LIN {X 0,Y 346.916,Z 553.438,A -85,B 0,C 180,E1 16644.293,E2 16644.293} C_VEL
LIN {X 0,Y 348.339,Z 562.311,A -85,B 0,C 180,E1 16644.634,E2 16644.634} C_VEL
LIN {X 0,Y 348.733,Z 569.969,A -85,B 0,C 180,E1 16644.843,E2 16644.843} C_VEL
LIN {X 0,Y 347.091,Z 583.273,A -85,B 0,C 180,E1 16645.017,E2 16645.017} C_VEL
LIN {X 0,Y 345.326,Z 596.669,A -85,B 0,C 180,E1 16645.186,E2 16645.186} C_VEL
LIN {X 0,Y 345.275,Z 597.789,A -85,B 0,C 180,E1 16645.208,E2 16645.208} C_VEL
LIN {X 0,Y 342.847,Z 683.726,A -85,B 0,C 180,E1 16647.121,E2 16647.121} C_VEL
LIN {X 0,Y 342.056,Z 700.444,A -85,B 0,C 180,E1 16647.822,E2 16647.822} C_VEL
LIN {X 0,Y 340.975,Z 714.968,A -85,B 0,C 180,E1 16648.731,E2 16648.731} C_VEL
LIN {X 0,Y 339.513,Z 729.938,A -85,B 0,C 180,E1 16650,E2 16650} C_VEL
LIN {X 0,Y 337.856,Z 743.563,A -85,B 0,C 180,E1 16651.526,E2 16651.526} C_VEL
LIN {X 0,Y 336.233,Z 755.603,A -85,B 0,C 180,E1 16653.239,E2 16653.239} C_VEL
LIN {X 0,Y 334.524,Z 767.051,A -85,B 0,C 180,E1 16655.316,E2 16655.316} C_VEL
LIN {X 0,Y 333.111,Z 776.185,A -85,B 0,C 180,E1 16657.415,E2 16657.415} C_VEL
LIN {X 0,Y 331.821,Z 784.518,A -85,B 0,C 180,E1 16659.89,E2 16659.89} C_VEL
LIN {X 0,Y 330.892,Z 790.802,A -85,B 0,C 180,E1 16662.388,E2 16662.388} C_VEL
LIN {X 0,Y 330.281,Z 795.59,A -85,B 0,C 180,E1 16665.09,E2 16665.09} C_VEL
LIN {X 0,Y 330.001,Z 798.505,A -85,B 0,C 180,E1 16667.819,E2 16667.819} C_VEL
LIN {X 0,Y 330.029,Z 799.71,A -85,B 0,C 180,E1 16670.584,E2 16670.584} C_VEL
LIN {X 0,Y 330.354,Z 799.125,A -85,B 0,C 180,E1 16673.359,E2 16673.359} C_VEL
LIN {X 0,Y 331.055,Z 796.754,A -85,B 0,C 180,E1 16676.164,E2 16676.164} C_VEL
LIN {X 0,Y 332.129,Z 792.619,A -85,B 0,C 180,E1 16678.83,E2 16678.83} C_VEL
LIN {X 0,Y 333.632,Z 786.717,A -85,B 0,C 180,E1 16681.43,E2 16681.43} C_VEL
LIN {X 0,Y 335.47,Z 779.072,A -85,B 0,C 180,E1 16683.872,E2 16683.872} C_VEL
LIN {X 0,Y 337.579,Z 769.937,A -85,B 0,C 180,E1 16686.115,E2 16686.115} C_VEL
LIN {X 0,Y 339.943,Z 758.678,A -85,B 0,C 180,E1 16688.249,E2 16688.249} C_VEL
LIN {X 0,Y 342.175,Z 746.843,A -85,B 0,C 180,E1 16690.005,E2 16690.005} C_VEL
LIN {X 0,Y 344.428,Z 733.255,A -85,B 0,C 180,E1 16691.58,E2 16691.58} C_VEL
LIN {X 0,Y 346.309,Z 719.123,A -85,B 0,C 180,E1 16692.832,E2 16692.832} C_VEL
LIN {X 0,Y 347.866,Z 703.791,A -85,B 0,C 180,E1 16693.844,E2 16693.844} C_VEL
LIN {X 0,Y 348.904,Z 687.638,A -85,B 0,C 180,E1 16694.564,E2 16694.564} C_VEL
LIN {X 0,Y 349.945,Z 659.796,A -85,B 0,C 180,E1 16695.275,E2 16695.275} C_VEL
LIN {X 0,Y 352.345,Z 591.836,A -85,B 0,C 180,E1 16696.795,E2 16696.795} C_VEL
LIN {X 0,Y 347.322,Z 564.262,A -85,B 0,C 180,E1 16698.138,E2 16698.138} C_VEL
LIN {X 0,Y 345.002,Z 552.728,A -85,B 0,C 180,E1 16698.806,E2 16698.806} C_VEL
LIN {X 0,Y 349.556,Z 526.788,A -85,B 0,C 180,E1 16703.353,E2 16703.353} C_VEL
LIN {X 0,Y 350.462,Z 522.011,A -85,B 0,C 180,E1 16704.206,E2 16704.206} C_VEL
LIN {X 0,Y 347.626,Z 509.823,A -85,B 0,C 180,E1 16707.266,E2 16707.266} C_VEL
LIN {X 0,Y 344.077,Z 497.71,A -85,B 0,C 180,E1 16710.665,E2 16710.665} C_VEL
LIN {X 0,Y 340.458,Z 487.061,A -85,B 0,C 180,E1 16714.05,E2 16714.05} C_VEL
LIN {X 0,Y 336.824,Z 477.501,A -85,B 0,C 180,E1 16717.484,E2 16717.484} C_VEL
LIN {X 0,Y 333.454,Z 469.646,A -85,B 0,C 180,E1 16720.741,E2 16720.741} C_VEL
LIN {X 0,Y 331.399,Z 465.22,A -85,B 0,C 180,E1 16722.802,E2 16722.802} C_VEL
LIN {X 0,Y 330.06,Z 461.809,A -85,B 0,C 180,E1 16724.539,E2 16724.539} C_VEL
LIN {X 0,Y 330.044,Z 461.676,A -85,B 0,C 180,E1 16728.82,E2 16728.82} C_VEL
LIN {X 0,Y 330.056,Z 461.676,A -85,B 0,C 180,E1 16733.215,E2 16733.215} C_VEL
LIN {X 0,Y 330.051,Z 461.685,A -85,B 0,C 180,E1 16737.569,E2 16737.569} C_VEL
LIN {X 0,Y 330.049,Z 461.686,A -85,B 0,C 180,E1 16741.909,E2 16741.909} C_VEL
LIN {X 0,Y 330.05,Z 461.673,A -85,B 0,C 180,E1 16746.261,E2 16746.261} C_VEL
LIN {X 0,Y 330.04,Z 461.665,A -85,B 0,C 180,E1 16750.649,E2 16750.649} C_VEL
LIN {X 0,Y 330.041,Z 461.658,A -85,B 0,C 180,E1 16754.922,E2 16754.922} C_VEL
LIN {X 0,Y 330.044,Z 461.659,A -85,B 0,C 180,E1 16759.281,E2 16759.281} C_VEL
LIN {X 0,Y 330.048,Z 461.661,A -85,B 0,C 180,E1 16763.571,E2 16763.571} C_VEL
LIN {X 0,Y 330.052,Z 461.662,A -85,B 0,C 180,E1 16768.005,E2 16768.005} C_VEL
LIN {X 0,Y 330.104,Z 462.019,A -85,B 0,C 180,E1 16770.785,E2 16770.785} C_VEL
LIN {X 0,Y 331.718,Z 465.65,A -85,B 0,C 180,E1 16772.447,E2 16772.447} C_VEL
LIN {X 0,Y 332.9,Z 468.27,A -85,B 0,C 180,E1 16773.548,E2 16773.548} C_VEL
LIN {X 0,Y 334.783,Z 471.961,A -85,B 0,C 180,E1 16775.083,E2 16775.083} C_VEL
LIN {X 0,Y 336.969,Z 476.649,A -85,B 0,C 180,E1 16776.825,E2 16776.825} C_VEL
LIN {X 0,Y 340.192,Z 483.549,A -85,B 0,C 180,E1 16779.191,E2 16779.191} C_VEL
LIN {X 0,Y 344.869,Z 494.751,A -85,B 0,C 180,E1 16782.494,E2 16782.494} C_VEL
LIN {X 0,Y 349.82,Z 507.787,A -85,B 0,C 180,E1 16785.781,E2 16785.781} C_VEL
LIN {X 0,Y 354.514,Z 522.198,A -85,B 0,C 180,E1 16788.918,E2 16788.918} C_VEL
LIN {X 0,Y 355.858,Z 526.854,A -85,B 0,C 180,E1 16789.839,E2 16789.839} C_VEL
LIN {X 0,Y 352.603,Z 543.562,A -85,B 0,C 180,E1 16791.896,E2 16791.896} C_VEL
LIN {X 0,Y 355.658,Z 572.916,A -85,B 0,C 180,E1 16793.022,E2 16793.022} C_VEL
LIN {X 0,Y 350.526,Z 732.105,A -85,B 0,C 180,E1 16796.34,E2 16796.34} C_VEL
LIN {X 0,Y 349.044,Z 750.459,A -85,B 0,C 180,E1 16796.989,E2 16796.989} C_VEL
LIN {X 0,Y 346.94,Z 768.318,A -85,B 0,C 180,E1 16797.918,E2 16797.918} C_VEL
LIN {X 0,Y 344.525,Z 784.972,A -85,B 0,C 180,E1 16799.091,E2 16799.091} C_VEL
LIN {X 0,Y 341.851,Z 801.23,A -85,B 0,C 180,E1 16800.569,E2 16800.569} C_VEL
LIN {X 0,Y 339.127,Z 816.442,A -85,B 0,C 180,E1 16802.305,E2 16802.305} C_VEL
LIN {X 0,Y 336.369,Z 831.077,A -85,B 0,C 180,E1 16804.365,E2 16804.365} C_VEL
LIN {X 0,Y 333.867,Z 844.636,A -85,B 0,C 180,E1 16806.715,E2 16806.715} C_VEL
LIN {X 0,Y 331.697,Z 857.019,A -85,B 0,C 180,E1 16809.349,E2 16809.349} C_VEL
LIN {X 0,Y 330.098,Z 867.902,A -85,B 0,C 180,E1 16812.186,E2 16812.186} C_VEL
LIN {X 0,Y 329.089,Z 877.24,A -85,B 0,C 180,E1 16815.214,E2 16815.214} C_VEL
LIN {X 0,Y 328.711,Z 884.849,A -85,B 0,C 180,E1 16818.362,E2 16818.362} C_VEL
LIN {X 0,Y 328.8,Z 890.405,A -85,B 0,C 180,E1 16821.431,E2 16821.431} C_VEL
LIN {X 0,Y 329.17,Z 894.144,A -85,B 0,C 180,E1 16824.422,E2 16824.422} C_VEL
LIN {X 0,Y 329.528,Z 896.232,A -85,B 0,C 180,E1 16827.392,E2 16827.392} C_VEL
LIN {X 0,Y 329.683,Z 896.689,A -85,B 0,C 180,E1 16830.174,E2 16830.174} C_VEL
LIN {X 0,Y 329.551,Z 895.671,A -85,B 0,C 180,E1 16832.957,E2 16832.957} C_VEL
LIN {X 0,Y 329.242,Z 893.161,A -85,B 0,C 180,E1 16835.752,E2 16835.752} C_VEL
LIN {X 0,Y 328.911,Z 888.783,A -85,B 0,C 180,E1 16838.743,E2 16838.743} C_VEL
LIN {X 0,Y 328.841,Z 882.577,A -85,B 0,C 180,E1 16841.755,E2 16841.755} C_VEL
LIN {X 0,Y 329.177,Z 874.384,A -85,B 0,C 180,E1 16844.783,E2 16844.783} C_VEL
LIN {X 0,Y 330.035,Z 864.634,A -85,B 0,C 180,E1 16847.636,E2 16847.636} C_VEL
LIN {X 0,Y 331.368,Z 853.376,A -85,B 0,C 180,E1 16850.304,E2 16850.304} C_VEL
LIN {X 0,Y 333.157,Z 840.616,A -85,B 0,C 180,E1 16852.778,E2 16852.778} C_VEL
LIN {X 0,Y 335.114,Z 827.266,A -85,B 0,C 180,E1 16854.903,E2 16854.903} C_VEL
LIN {X 0,Y 337.383,Z 812.153,A -85,B 0,C 180,E1 16856.87,E2 16856.87} C_VEL
LIN {X 0,Y 339.644,Z 796.004,A -85,B 0,C 180,E1 16858.554,E2 16858.554} C_VEL
LIN {X 0,Y 341.821,Z 778.87,A -85,B 0,C 180,E1 16859.956,E2 16859.956} C_VEL
LIN {X 0,Y 343.792,Z 760.66,A -85,B 0,C 180,E1 16861.08,E2 16861.08} C_VEL
LIN {X 0,Y 345.324,Z 742.426,A -85,B 0,C 180,E1 16861.874,E2 16861.874} C_VEL
LIN {X 0,Y 346.161,Z 723.688,A -85,B 0,C 180,E1 16862.394,E2 16862.394} C_VEL
LIN {X 0,Y 349.848,Z 570.703,A -85,B 0,C 180,E1 16865.478,E2 16865.478} C_VEL
LIN {X 0,Y 347.149,Z 542.148,A -85,B 0,C 180,E1 16866.393,E2 16866.393} C_VEL
LIN {X 0,Y 350.527,Z 520.086,A -85,B 0,C 180,E1 16869.059,E2 16869.059} C_VEL
LIN {X 0,Y 344.365,Z 500.623,A -85,B 0,C 180,E1 16872.483,E2 16872.483} C_VEL
LIN {X 0,Y 337.938,Z 482.37,A -85,B 0,C 180,E1 16876.067,E2 16876.067} C_VEL
LIN {X 0,Y 332.331,Z 467.887,A -85,B 0,C 180,E1 16879.242,E2 16879.242} C_VEL
LIN {X 0,Y 330.059,Z 461.834,A -85,B 0,C 180,E1 16880.719,E2 16880.719} C_VEL
LIN {X 0,Y 330.043,Z 461.675,A -85,B 0,C 180,E1 16885.07,E2 16885.07} C_VEL
LIN {X 0,Y 330.057,Z 461.674,A -85,B 0,C 180,E1 16889.408,E2 16889.408} C_VEL
LIN {X 0,Y 330.051,Z 461.664,A -85,B 0,C 180,E1 16893.75,E2 16893.75} C_VEL
LIN {X 0,Y 330.052,Z 461.657,A -85,B 0,C 180,E1 16898.123,E2 16898.123} C_VEL
LIN {X 0,Y 330.033,Z 461.68,A -85,B 0,C 180,E1 16902.547,E2 16902.547} C_VEL
LIN {X 0,Y 330.027,Z 461.676,A -85,B 0,C 180,E1 16906.867,E2 16906.867} C_VEL
LIN {X 0,Y 330.02,Z 461.653,A -85,B 0,C 180,E1 16911.287,E2 16911.287} C_VEL
LIN {X 0,Y 330.025,Z 461.687,A -85,B 0,C 180,E1 16915.482,E2 16915.482} C_VEL
LIN {X 0,Y 330.03,Z 461.642,A -85,B 0,C 180,E1 16919.827,E2 16919.827} C_VEL
LIN {X 0,Y 330.041,Z 461.684,A -85,B 0,C 180,E1 16924.17,E2 16924.17} C_VEL
LIN {X 0,Y 330.038,Z 461.638,A -85,B 0,C 180,E1 16928.537,E2 16928.537} C_VEL
LIN {X 0,Y 330.022,Z 461.689,A -85,B 0,C 180,E1 16932.956,E2 16932.956} C_VEL
LIN {X 0,Y 330.012,Z 461.64,A -85,B 0,C 180,E1 16937.091,E2 16937.091} C_VEL
LIN {X 0,Y 330.009,Z 461.69,A -85,B 0,C 180,E1 16941.32,E2 16941.32} C_VEL
LIN {X 0,Y 329.998,Z 461.647,A -85,B 0,C 180,E1 16945.676,E2 16945.676} C_VEL
LIN {X 0,Y 330.003,Z 461.69,A -85,B 0,C 180,E1 16949.996,E2 16949.996} C_VEL
LIN {X 0,Y 330.001,Z 461.65,A -85,B 0,C 180,E1 16954.303,E2 16954.303} C_VEL
LIN {X 0,Y 330.017,Z 461.688,A -85,B 0,C 180,E1 16958.618,E2 16958.618} C_VEL
LIN {X 0,Y 330.018,Z 461.668,A -85,B 0,C 180,E1 16962.845,E2 16962.845} C_VEL
LIN {X 0,Y 330.014,Z 461.663,A -85,B 0,C 180,E1 16967.26,E2 16967.26} C_VEL
LIN {X 0,Y 330.012,Z 461.683,A -85,B 0,C 180,E1 16971.415,E2 16971.415} C_VEL
LIN {X 0,Y 329.989,Z 461.692,A -85,B 0,C 180,E1 16975.811,E2 16975.811} C_VEL
LIN {X 0,Y 329.983,Z 461.694,A -85,B 0,C 180,E1 16980.066,E2 16980.066} C_VEL
LIN {X 0,Y 329.986,Z 461.695,A -85,B 0,C 180,E1 16984.323,E2 16984.323} C_VEL
LIN {X 0,Y 330.075,Z 462.225,A -85,B 0,C 180,E1 16984.715,E2 16984.715} C_VEL
LIN {X 0,Y 334.332,Z 474.661,A -85,B 0,C 180,E1 16988.048,E2 16988.048} C_VEL
LIN {X 0,Y 338.877,Z 489.203,A -85,B 0,C 180,E1 16991.596,E2 16991.596} C_VEL
LIN {X 0,Y 343.127,Z 504.85,A -85,B 0,C 180,E1 16995.141,E2 16995.141} C_VEL
LIN {X 0,Y 344.958,Z 513.335,A -85,B 0,C 180,E1 16996.933,E2 16996.933} C_VEL
LIN {X 0,Y 341.225,Z 539.64,A -85,B 0,C 180,E1 17001.405,E2 17001.405} C_VEL
LIN {X 0,Y 339.552,Z 552.539,A -85,B 0,C 180,E1 17003.575,E2 17003.575} C_VEL
LIN {X 0,Y 339.887,Z 555.622,A -85,B 0,C 180,E1 17003.767,E2 17003.767} C_VEL
LIN {X 0,Y 345.466,Z 591.168,A -85,B 0,C 180,E1 17005.069,E2 17005.069} C_VEL
LIN {X 0,Y 345.275,Z 597.789,A -85,B 0,C 180,E1 17005.208,E2 17005.208} C_VEL
LIN {X 0,Y 344.122,Z 605.458,A -85,B 0,C 180,E1 17005.293,E2 17005.293} C_VEL
LIN {X 0,Y 337.892,Z 625.774,A -85,B 0,C 180,E1 17005.272,E2 17005.272} C_VEL
LIN {X 0,Y 337.059,Z 632.354,A -85,B 0,C 180,E1 17005.364,E2 17005.364} C_VEL
LIN {X 0,Y 335.511,Z 685.056,A -85,B 0,C 180,E1 17006.604,E2 17006.604} C_VEL
LIN {X 0,Y 334.705,Z 701.246,A -85,B 0,C 180,E1 17007.303,E2 17007.303} C_VEL
LIN {X 0,Y 333.515,Z 716.419,A -85,B 0,C 180,E1 17008.282,E2 17008.282} C_VEL
LIN {X 0,Y 332.102,Z 730.276,A -85,B 0,C 180,E1 17009.482,E2 17009.482} C_VEL
LIN {X 0,Y 330.372,Z 744.029,A -85,B 0,C 180,E1 17011.04,E2 17011.04} C_VEL
LIN {X 0,Y 328.67,Z 756.171,A -85,B 0,C 180,E1 17012.79,E2 17012.79} C_VEL
LIN {X 0,Y 326.874,Z 767.702,A -85,B 0,C 180,E1 17014.913,E2 17014.913} C_VEL
LIN {X 0,Y 325.388,Z 776.93,A -85,B 0,C 180,E1 17017.06,E2 17017.06} C_VEL
LIN {X 0,Y 324.024,Z 785.331,A -85,B 0,C 180,E1 17019.592,E2 17019.592} C_VEL
LIN {X 0,Y 323.041,Z 791.706,A -85,B 0,C 180,E1 17022.15,E2 17022.15} C_VEL
LIN {X 0,Y 322.386,Z 796.564,A -85,B 0,C 180,E1 17024.917,E2 17024.917} C_VEL
LIN {X 0,Y 322.087,Z 799.578,A -85,B 0,C 180,E1 17027.711,E2 17027.711} C_VEL
LIN {X 0,Y 322.124,Z 800.896,A -85,B 0,C 180,E1 17030.723,E2 17030.723} C_VEL
LIN {X 0,Y 322.488,Z 800.291,A -85,B 0,C 180,E1 17033.575,E2 17033.575} C_VEL
LIN {X 0,Y 323.255,Z 797.911,A -85,B 0,C 180,E1 17036.449,E2 17036.449} C_VEL
LIN {X 0,Y 324.478,Z 793.539,A -85,B 0,C 180,E1 17039.302,E2 17039.302} C_VEL
LIN {X 0,Y 326.03,Z 787.855,A -85,B 0,C 180,E1 17041.842,E2 17041.842} C_VEL
LIN {X 0,Y 327.984,Z 780.248,A -85,B 0,C 180,E1 17044.331,E2 17044.331} C_VEL
LIN {X 0,Y 330.256,Z 771.024,A -85,B 0,C 180,E1 17046.649,E2 17046.649} C_VEL
LIN {X 0,Y 332.725,Z 759.971,A -85,B 0,C 180,E1 17048.796,E2 17048.796} C_VEL
LIN {X 0,Y 335.078,Z 748.293,A -85,B 0,C 180,E1 17050.579,E2 17050.579} C_VEL
LIN {X 0,Y 337.549,Z 734.162,A -85,B 0,C 180,E1 17052.252,E2 17052.252} C_VEL
LIN {X 0,Y 339.57,Z 719.702,A -85,B 0,C 180,E1 17053.551,E2 17053.551} C_VEL
LIN {X 0,Y 341.145,Z 704.969,A -85,B 0,C 180,E1 17054.54,E2 17054.54} C_VEL
LIN {X 0,Y 342.244,Z 689.079,A -85,B 0,C 180,E1 17055.273,E2 17055.273} C_VEL
LIN {X 0,Y 343.175,Z 665.403,A -85,B 0,C 180,E1 17055.909,E2 17055.909} C_VEL
LIN {X 0,Y 345.891,Z 593.204,A -85,B 0,C 180,E1 17057.552,E2 17057.552} C_VEL
LIN {X 0,Y 341.017,Z 566.089,A -85,B 0,C 180,E1 17058.918,E2 17058.918} C_VEL
LIN {X 0,Y 338.291,Z 552.635,A -85,B 0,C 180,E1 17059.713,E2 17059.713} C_VEL
LIN {X 0,Y 343.163,Z 526.668,A -85,B 0,C 180,E1 17064.357,E2 17064.357} C_VEL
LIN {X 0,Y 343.366,Z 524.479,A -85,B 0,C 180,E1 17064.79,E2 17064.79} C_VEL
LIN {X 0,Y 340.545,Z 512.512,A -85,B 0,C 180,E1 17067.898,E2 17067.898} C_VEL
LIN {X 0,Y 337.184,Z 500.875,A -85,B 0,C 180,E1 17071.289,E2 17071.289} C_VEL
LIN {X 0,Y 333.719,Z 490.759,A -85,B 0,C 180,E1 17074.631,E2 17074.631} C_VEL
LIN {X 0,Y 330.529,Z 482.269,A -85,B 0,C 180,E1 17077.782,E2 17077.782} C_VEL
LIN {X 0,Y 327.447,Z 474.847,A -85,B 0,C 180,E1 17080.929,E2 17080.929} C_VEL
LIN {X 0,Y 325.445,Z 470.463,A -85,B 0,C 180,E1 17083.03,E2 17083.03} C_VEL
LIN {X 0,Y 323.624,Z 466.427,A -85,B 0,C 180,E1 17085.141,E2 17085.141} C_VEL
LIN {X 0,Y 322.129,Z 462.79,A -85,B 0,C 180,E1 17087.268,E2 17087.268} C_VEL
LIN {X 0,Y 322.111,Z 462.66,A -85,B 0,C 180,E1 17091.79,E2 17091.79} C_VEL
LIN {X 0,Y 322.101,Z 462.659,A -85,B 0,C 180,E1 17096.262,E2 17096.262} C_VEL
LIN {X 0,Y 322.099,Z 462.653,A -85,B 0,C 180,E1 17100.711,E2 17100.711} C_VEL
LIN {X 0,Y 322.104,Z 462.647,A -85,B 0,C 180,E1 17105.164,E2 17105.164} C_VEL
LIN {X 0,Y 322.107,Z 462.645,A -85,B 0,C 180,E1 17109.469,E2 17109.469} C_VEL
LIN {X 0,Y 322.112,Z 462.647,A -85,B 0,C 180,E1 17113.828,E2 17113.828} C_VEL
LIN {X 0,Y 322.11,Z 462.653,A -85,B 0,C 180,E1 17118.271,E2 17118.271} C_VEL
LIN {X 0,Y 322.112,Z 462.658,A -85,B 0,C 180,E1 17122.638,E2 17122.638} C_VEL
LIN {X 0,Y 322.105,Z 462.657,A -85,B 0,C 180,E1 17127.149,E2 17127.149} C_VEL
LIN {X 0,Y 322.202,Z 463.203,A -85,B 0,C 180,E1 17128.144,E2 17128.144} C_VEL
LIN {X 0,Y 324.057,Z 466.996,A -85,B 0,C 180,E1 17130.194,E2 17130.194} C_VEL
LIN {X 0,Y 326.958,Z 472.923,A -85,B 0,C 180,E1 17132.979,E2 17132.979} C_VEL
LIN {X 0,Y 329.255,Z 477.888,A -85,B 0,C 180,E1 17135.025,E2 17135.025} C_VEL
LIN {X 0,Y 332.561,Z 484.777,A -85,B 0,C 180,E1 17137.613,E2 17137.613} C_VEL
LIN {X 0,Y 337.276,Z 495.909,A -85,B 0,C 180,E1 17141.157,E2 17141.157} C_VEL
LIN {X 0,Y 342.098,Z 508.445,A -85,B 0,C 180,E1 17144.544,E2 17144.544} C_VEL
LIN {X 0,Y 346.518,Z 521.675,A -85,B 0,C 180,E1 17147.618,E2 17147.618} C_VEL
LIN {X 0,Y 348.913,Z 530.051,A -85,B 0,C 180,E1 17149.362,E2 17149.362} C_VEL
LIN {X 0,Y 346.123,Z 543.724,A -85,B 0,C 180,E1 17151.067,E2 17151.067} C_VEL
LIN {X 0,Y 349.173,Z 573.441,A -85,B 0,C 180,E1 17152.249,E2 17152.249} C_VEL
LIN {X 0,Y 343.844,Z 731.353,A -85,B 0,C 180,E1 17155.602,E2 17155.602} C_VEL
LIN {X 0,Y 342.304,Z 749.658,A -85,B 0,C 180,E1 17156.259,E2 17156.259} C_VEL
LIN {X 0,Y 340.191,Z 766.866,A -85,B 0,C 180,E1 17157.162,E2 17157.162} C_VEL
LIN {X 0,Y 337.587,Z 784.01,A -85,B 0,C 180,E1 17158.384,E2 17158.384} C_VEL
LIN {X 0,Y 334.775,Z 800.275,A -85,B 0,C 180,E1 17159.884,E2 17159.884} C_VEL
LIN {X 0,Y 331.876,Z 815.674,A -85,B 0,C 180,E1 17161.673,E2 17161.673} C_VEL
LIN {X 0,Y 328.981,Z 830.167,A -85,B 0,C 180,E1 17163.755,E2 17163.755} C_VEL
LIN {X 0,Y 326.328,Z 843.652,A -85,B 0,C 180,E1 17166.144,E2 17166.144} C_VEL
LIN {X 0,Y 324.008,Z 856.018,A -85,B 0,C 180,E1 17168.836,E2 17168.836} C_VEL
LIN {X 0,Y 322.279,Z 866.853,A -85,B 0,C 180,E1 17171.739,E2 17171.739} C_VEL
LIN {X 0,Y 321.17,Z 876.152,A -85,B 0,C 180,E1 17174.841,E2 17174.841} C_VEL
LIN {X 0,Y 320.744,Z 883.488,A -85,B 0,C 180,E1 17177.945,E2 17177.945} C_VEL
LIN {X 0,Y 320.805,Z 889.133,A -85,B 0,C 180,E1 17181.113,E2 17181.113} C_VEL
LIN {X 0,Y 321.203,Z 893.015,A -85,B 0,C 180,E1 17184.284,E2 17184.284} C_VEL
LIN {X 0,Y 321.581,Z 894.998,A -85,B 0,C 180,E1 17187.149,E2 17187.149} C_VEL
LIN {X 0,Y 321.774,Z 895.523,A -85,B 0,C 180,E1 17190,E2 17190} C_VEL
LIN {X 0,Y 321.643,Z 894.559,A -85,B 0,C 180,E1 17192.851,E2 17192.851} C_VEL
LIN {X 0,Y 321.314,Z 892.091,A -85,B 0,C 180,E1 17195.715,E2 17195.715} C_VEL
LIN {X 0,Y 320.957,Z 887.749,A -85,B 0,C 180,E1 17198.781,E2 17198.781} C_VEL
LIN {X 0,Y 320.877,Z 881.443,A -85,B 0,C 180,E1 17201.923,E2 17201.923} C_VEL
LIN {X 0,Y 321.226,Z 873.406,A -85,B 0,C 180,E1 17204.972,E2 17204.972} C_VEL
LIN {X 0,Y 322.128,Z 863.68,A -85,B 0,C 180,E1 17207.896,E2 17207.896} C_VEL
LIN {X 0,Y 323.522,Z 852.442,A -85,B 0,C 180,E1 17210.63,E2 17210.63} C_VEL
LIN {X 0,Y 325.391,Z 839.689,A -85,B 0,C 180,E1 17213.161,E2 17213.161} C_VEL
LIN {X 0,Y 327.497,Z 825.938,A -85,B 0,C 180,E1 17215.392,E2 17215.392} C_VEL
LIN {X 0,Y 329.801,Z 811.17,A -85,B 0,C 180,E1 17217.341,E2 17217.341} C_VEL
LIN {X 0,Y 332.153,Z 794.919,A -85,B 0,C 180,E1 17219.064,E2 17219.064} C_VEL
LIN {X 0,Y 334.353,Z 778.274,A -85,B 0,C 180,E1 17220.452,E2 17220.452} C_VEL
LIN {X 0,Y 336.38,Z 760.196,A -85,B 0,C 180,E1 17221.594,E2 17221.594} C_VEL
LIN {X 0,Y 337.977,Z 741.833,A -85,B 0,C 180,E1 17222.411,E2 17222.411} C_VEL
LIN {X 0,Y 338.842,Z 723.112,A -85,B 0,C 180,E1 17222.942,E2 17222.942} C_VEL
LIN {X 0,Y 342.691,Z 571.617,A -85,B 0,C 180,E1 17226.054,E2 17226.054} C_VEL
LIN {X 0,Y 339.983,Z 542.148,A -85,B 0,C 180,E1 17227.024,E2 17227.024} C_VEL
LIN {X 0,Y 343.146,Z 522.552,A -85,B 0,C 180,E1 17229.452,E2 17229.452} C_VEL
LIN {X 0,Y 337.112,Z 503.455,A -85,B 0,C 180,E1 17232.896,E2 17232.896} C_VEL
LIN {X 0,Y 330.958,Z 485.681,A -85,B 0,C 180,E1 17236.475,E2 17236.475} C_VEL
LIN {X 0,Y 324.993,Z 470.069,A -85,B 0,C 180,E1 17240.002,E2 17240.002} C_VEL
LIN {X 0,Y 322.138,Z 462.852,A -85,B 0,C 180,E1 17241.839,E2 17241.839} C_VEL
LIN {X 0,Y 322.109,Z 462.677,A -85,B 0,C 180,E1 17246.032,E2 17246.032} C_VEL
LIN {X 0,Y 322.1,Z 462.678,A -85,B 0,C 180,E1 17250.425,E2 17250.425} C_VEL
LIN {X 0,Y 322.094,Z 462.671,A -85,B 0,C 180,E1 17254.832,E2 17254.832} C_VEL
LIN {X 0,Y 322.097,Z 462.651,A -85,B 0,C 180,E1 17259.275,E2 17259.275} C_VEL
LIN {X 0,Y 322.104,Z 462.649,A -85,B 0,C 180,E1 17263.592,E2 17263.592} C_VEL
LIN {X 0,Y 322.111,Z 462.674,A -85,B 0,C 180,E1 17267.997,E2 17267.997} C_VEL
LIN {X 0,Y 322.106,Z 462.634,A -85,B 0,C 180,E1 17272.33,E2 17272.33} C_VEL
LIN {X 0,Y 322.093,Z 462.674,A -85,B 0,C 180,E1 17276.619,E2 17276.619} C_VEL
LIN {X 0,Y 322.079,Z 462.634,A -85,B 0,C 180,E1 17280.89,E2 17280.89} C_VEL
LIN {X 0,Y 322.076,Z 462.672,A -85,B 0,C 180,E1 17285.344,E2 17285.344} C_VEL
LIN {X 0,Y 322.072,Z 462.634,A -85,B 0,C 180,E1 17289.651,E2 17289.651} C_VEL
LIN {X 0,Y 322.085,Z 462.676,A -85,B 0,C 180,E1 17294.013,E2 17294.013} C_VEL
LIN {X 0,Y 322.093,Z 462.629,A -85,B 0,C 180,E1 17298.46,E2 17298.46} C_VEL
LIN {X 0,Y 322.098,Z 462.671,A -85,B 0,C 180,E1 17302.832,E2 17302.832} C_VEL
LIN {X 0,Y 322.075,Z 462.637,A -85,B 0,C 180,E1 17307.152,E2 17307.152} C_VEL
LIN {X 0,Y 322.066,Z 462.673,A -85,B 0,C 180,E1 17311.437,E2 17311.437} C_VEL
LIN {X 0,Y 322.053,Z 462.656,A -85,B 0,C 180,E1 17315.873,E2 17315.873} C_VEL
LIN {X 0,Y 322.053,Z 462.655,A -85,B 0,C 180,E1 17320.224,E2 17320.224} C_VEL
LIN {X 0,Y 322.064,Z 462.68,A -85,B 0,C 180,E1 17324.558,E2 17324.558} C_VEL
LIN {X 0,Y 322.084,Z 462.66,A -85,B 0,C 180,E1 17329.079,E2 17329.079} C_VEL
LIN {X 0,Y 322.068,Z 462.657,A -85,B 0,C 180,E1 17333.411,E2 17333.411} C_VEL
LIN {X 0,Y 322.056,Z 462.661,A -85,B 0,C 180,E1 17337.724,E2 17337.724} C_VEL
LIN {X 0,Y 322.047,Z 462.666,A -85,B 0,C 180,E1 17342.043,E2 17342.043} C_VEL
LIN {X 0,Y 322.118,Z 462.988,A -85,B 0,C 180,E1 17343.574,E2 17343.574} C_VEL
LIN {X 0,Y 326.747,Z 476.437,A -85,B 0,C 180,E1 17347.321,E2 17347.321} C_VEL
LIN {X 0,Y 331.273,Z 490.987,A -85,B 0,C 180,E1 17350.975,E2 17350.975} C_VEL
LIN {X 0,Y 335.302,Z 505.799,A -85,B 0,C 180,E1 17354.432,E2 17354.432} C_VEL
LIN {X 0,Y 337.56,Z 515.497,A -85,B 0,C 180,E1 17356.554,E2 17356.554} C_VEL
LIN {X 0,Y 333.591,Z 542.414,A -85,B 0,C 180,E1 17361.207,E2 17361.207} C_VEL
LIN {X 0,Y 332.208,Z 553.269,A -85,B 0,C 180,E1 17363.013,E2 17363.013} C_VEL
LIN {X 0,Y 338.266,Z 592.213,A -85,B 0,C 180,E1 17364.495,E2 17364.495} C_VEL
LIN {X 0,Y 337.059,Z 632.354,A -85,B 0,C 180,E1 17365.364,E2 17365.364} C_VEL
LIN {X 0,Y 335.972,Z 640.016,A -85,B 0,C 180,E1 17365.462,E2 17365.462} C_VEL
LIN {X 0,Y 329.69,Z 660.32,A -85,B 0,C 180,E1 17365.455,E2 17365.455} C_VEL
LIN {X 0,Y 328.783,Z 666.9,A -85,B 0,C 180,E1 17365.549,E2 17365.549} C_VEL
LIN {X 0,Y 328.108,Z 688.799,A -85,B 0,C 180,E1 17366.15,E2 17366.15} C_VEL
LIN {X 0,Y 327.218,Z 704.301,A -85,B 0,C 180,E1 17366.891,E2 17366.891} C_VEL
LIN {X 0,Y 325.877,Z 720.004,A -85,B 0,C 180,E1 17367.978,E2 17367.978} C_VEL
LIN {X 0,Y 324.198,Z 734.81,A -85,B 0,C 180,E1 17369.381,E2 17369.381} C_VEL
LIN {X 0,Y 322.404,Z 748.144,A -85,B 0,C 180,E1 17371.02,E2 17371.02} C_VEL
LIN {X 0,Y 320.464,Z 760.908,A -85,B 0,C 180,E1 17373.04,E2 17373.04} C_VEL
LIN {X 0,Y 318.684,Z 771.677,A -85,B 0,C 180,E1 17375.22,E2 17375.22} C_VEL
LIN {X 0,Y 317.12,Z 780.961,A -85,B 0,C 180,E1 17377.609,E2 17377.609} C_VEL
LIN {X 0,Y 315.819,Z 788.661,A -85,B 0,C 180,E1 17380.212,E2 17380.212} C_VEL
LIN {X 0,Y 314.903,Z 794.581,A -85,B 0,C 180,E1 17382.896,E2 17382.896} C_VEL
LIN {X 0,Y 314.321,Z 798.992,A -85,B 0,C 180,E1 17385.876,E2 17385.876} C_VEL
LIN {X 0,Y 314.141,Z 801.404,A -85,B 0,C 180,E1 17388.751,E2 17388.751} C_VEL
LIN {X 0,Y 314.314,Z 802.065,A -85,B 0,C 180,E1 17391.85,E2 17391.85} C_VEL
LIN {X 0,Y 314.853,Z 800.864,A -85,B 0,C 180,E1 17394.783,E2 17394.783} C_VEL
LIN {X 0,Y 315.849,Z 797.827,A -85,B 0,C 180,E1 17397.732,E2 17397.732} C_VEL
LIN {X 0,Y 317.259,Z 793.107,A -85,B 0,C 180,E1 17400.49,E2 17400.49} C_VEL
LIN {X 0,Y 319.19,Z 786.406,A -85,B 0,C 180,E1 17403.242,E2 17403.242} C_VEL
LIN {X 0,Y 321.463,Z 777.968,A -85,B 0,C 180,E1 17405.785,E2 17405.785} C_VEL
LIN {X 0,Y 323.779,Z 768.88,A -85,B 0,C 180,E1 17407.917,E2 17407.917} C_VEL
LIN {X 0,Y 326.3,Z 757.857,A -85,B 0,C 180,E1 17409.949,E2 17409.949} C_VEL
LIN {X 0,Y 328.858,Z 745.476,A -85,B 0,C 180,E1 17411.747,E2 17411.747} C_VEL
LIN {X 0,Y 331.2,Z 732.038,A -85,B 0,C 180,E1 17413.258,E2 17413.258} C_VEL
LIN {X 0,Y 333.196,Z 717.939,A -85,B 0,C 180,E1 17414.483,E2 17414.483} C_VEL
LIN {X 0,Y 334.789,Z 702.528,A -85,B 0,C 180,E1 17415.463,E2 17415.463} C_VEL
LIN {X 0,Y 335.876,Z 686.24,A -85,B 0,C 180,E1 17416.164,E2 17416.164} C_VEL
LIN {X 0,Y 339.389,Z 601.216,A -85,B 0,C 180,E1 17418.165,E2 17418.165} C_VEL
LIN {X 0,Y 339.456,Z 594.283,A -85,B 0,C 180,E1 17418.35,E2 17418.35} C_VEL
LIN {X 0,Y 334.512,Z 566.405,A -85,B 0,C 180,E1 17419.815,E2 17419.815} C_VEL
LIN {X 0,Y 331.715,Z 552.565,A -85,B 0,C 180,E1 17420.673,E2 17420.673} C_VEL
LIN {X 0,Y 336.517,Z 528.22,A -85,B 0,C 180,E1 17425.089,E2 17425.089} C_VEL
LIN {X 0,Y 333.707,Z 515.937,A -85,B 0,C 180,E1 17428.376,E2 17428.376} C_VEL
LIN {X 0,Y 330.577,Z 504.974,A -85,B 0,C 180,E1 17431.66,E2 17431.66} C_VEL
LIN {X 0,Y 327.217,Z 494.922,A -85,B 0,C 180,E1 17435.059,E2 17435.059} C_VEL
LIN {X 0,Y 324.094,Z 486.642,A -85,B 0,C 180,E1 17438.271,E2 17438.271} C_VEL
LIN {X 0,Y 321.457,Z 480.058,A -85,B 0,C 180,E1 17441.126,E2 17441.126} C_VEL
LIN {X 0,Y 319.51,Z 475.71,A -85,B 0,C 180,E1 17443.267,E2 17443.267} C_VEL
LIN {X 0,Y 317.903,Z 471.993,A -85,B 0,C 180,E1 17445.24,E2 17445.24} C_VEL
LIN {X 0,Y 315.947,Z 467.782,A -85,B 0,C 180,E1 17447.758,E2 17447.758} C_VEL
LIN {X 0,Y 314.177,Z 463.759,A -85,B 0,C 180,E1 17450.659,E2 17450.659} C_VEL
LIN {X 0,Y 314.166,Z 463.636,A -85,B 0,C 180,E1 17455.07,E2 17455.07} C_VEL
LIN {X 0,Y 314.173,Z 463.633,A -85,B 0,C 180,E1 17459.453,E2 17459.453} C_VEL
LIN {X 0,Y 314.168,Z 463.636,A -85,B 0,C 180,E1 17463.832,E2 17463.832} C_VEL
LIN {X 0,Y 314.172,Z 463.643,A -85,B 0,C 180,E1 17468.233,E2 17468.233} C_VEL
LIN {X 0,Y 314.165,Z 463.653,A -85,B 0,C 180,E1 17472.685,E2 17472.685} C_VEL
LIN {X 0,Y 314.168,Z 463.662,A -85,B 0,C 180,E1 17477.216,E2 17477.216} C_VEL
LIN {X 0,Y 314.178,Z 463.664,A -85,B 0,C 180,E1 17481.678,E2 17481.678} C_VEL
LIN {X 0,Y 314.217,Z 463.972,A -85,B 0,C 180,E1 17484.706,E2 17484.706} C_VEL
LIN {X 0,Y 316.102,Z 467.956,A -85,B 0,C 180,E1 17487.3,E2 17487.3} C_VEL
LIN {X 0,Y 317.03,Z 469.974,A -85,B 0,C 180,E1 17488.439,E2 17488.439} C_VEL
LIN {X 0,Y 319.079,Z 473.698,A -85,B 0,C 180,E1 17490.506,E2 17490.506} C_VEL
LIN {X 0,Y 321.518,Z 479.023,A -85,B 0,C 180,E1 17492.971,E2 17492.971} C_VEL
LIN {X 0,Y 323.617,Z 483.512,A -85,B 0,C 180,E1 17494.86,E2 17494.86} C_VEL
LIN {X 0,Y 326.832,Z 490.478,A -85,B 0,C 180,E1 17497.502,E2 17497.502} C_VEL
LIN {X 0,Y 331.26,Z 501.011,A -85,B 0,C 180,E1 17500.918,E2 17500.918} C_VEL
LIN {X 0,Y 335.724,Z 512.811,A -85,B 0,C 180,E1 17504.179,E2 17504.179} C_VEL
LIN {X 0,Y 340.022,Z 525.986,A -85,B 0,C 180,E1 17507.319,E2 17507.319} C_VEL
LIN {X 0,Y 341.976,Z 533.304,A -85,B 0,C 180,E1 17508.864,E2 17508.864} C_VEL
LIN {X 0,Y 339.715,Z 543.942,A -85,B 0,C 180,E1 17510.209,E2 17510.209} C_VEL
LIN {X 0,Y 342.755,Z 573.863,A -85,B 0,C 180,E1 17511.441,E2 17511.441} C_VEL
LIN {X 0,Y 337.23,Z 730.703,A -85,B 0,C 180,E1 17514.834,E2 17514.834} C_VEL
LIN {X 0,Y 335.629,Z 749.007,A -85,B 0,C 180,E1 17515.501,E2 17515.501} C_VEL
LIN {X 0,Y 333.435,Z 766.098,A -85,B 0,C 180,E1 17516.41,E2 17516.41} C_VEL
LIN {X 0,Y 330.717,Z 783.226,A -85,B 0,C 180,E1 17517.648,E2 17517.648} C_VEL
LIN {X 0,Y 327.76,Z 799.422,A -85,B 0,C 180,E1 17519.17,E2 17519.17} C_VEL
LIN {X 0,Y 324.714,Z 814.72,A -85,B 0,C 180,E1 17520.984,E2 17520.984} C_VEL
LIN {X 0,Y 321.528,Z 829.75,A -85,B 0,C 180,E1 17523.198,E2 17523.198} C_VEL
LIN {X 0,Y 318.824,Z 842.667,A -85,B 0,C 180,E1 17525.546,E2 17525.546} C_VEL
LIN {X 0,Y 316.345,Z 855.015,A -85,B 0,C 180,E1 17528.297,E2 17528.297} C_VEL
LIN {X 0,Y 314.425,Z 866.172,A -85,B 0,C 180,E1 17531.374,E2 17531.374} C_VEL
LIN {X 0,Y 313.229,Z 875.456,A -85,B 0,C 180,E1 17534.582,E2 17534.582} C_VEL
LIN {X 0,Y 312.761,Z 882.786,A -85,B 0,C 180,E1 17537.82,E2 17537.82} C_VEL
LIN {X 0,Y 312.841,Z 888.461,A -85,B 0,C 180,E1 17541.176,E2 17541.176} C_VEL
LIN {X 0,Y 313.289,Z 892.23,A -85,B 0,C 180,E1 17544.506,E2 17544.506} C_VEL
LIN {X 0,Y 313.7,Z 894.088,A -85,B 0,C 180,E1 17547.626,E2 17547.626} C_VEL
LIN {X 0,Y 313.849,Z 894.283,A -85,B 0,C 180,E1 17550.548,E2 17550.548} C_VEL
LIN {X 0,Y 313.671,Z 892.971,A -85,B 0,C 180,E1 17553.473,E2 17553.473} C_VEL
LIN {X 0,Y 313.286,Z 890.134,A -85,B 0,C 180,E1 17556.414,E2 17556.414} C_VEL
LIN {X 0,Y 312.952,Z 885.409,A -85,B 0,C 180,E1 17559.564,E2 17559.564} C_VEL
LIN {X 0,Y 312.947,Z 878.827,A -85,B 0,C 180,E1 17562.736,E2 17562.736} C_VEL
LIN {X 0,Y 313.411,Z 870.775,A -85,B 0,C 180,E1 17565.734,E2 17565.734} C_VEL
LIN {X 0,Y 314.465,Z 860.668,A -85,B 0,C 180,E1 17568.732,E2 17568.732} C_VEL
LIN {X 0,Y 316.062,Z 848.952,A -85,B 0,C 180,E1 17571.529,E2 17571.529} C_VEL
LIN {X 0,Y 318.053,Z 836.11,A -85,B 0,C 180,E1 17574.024,E2 17574.024} C_VEL
LIN {X 0,Y 320.354,Z 821.699,A -85,B 0,C 180,E1 17576.308,E2 17576.308} C_VEL
LIN {X 0,Y 322.831,Z 806.276,A -85,B 0,C 180,E1 17578.286,E2 17578.286} C_VEL
LIN {X 0,Y 325.268,Z 789.85,A -85,B 0,C 180,E1 17579.968,E2 17579.968} C_VEL
LIN {X 0,Y 327.434,Z 773.559,A -85,B 0,C 180,E1 17581.273,E2 17581.273} C_VEL
LIN {X 0,Y 329.453,Z 755.496,A -85,B 0,C 180,E1 17582.359,E2 17582.359} C_VEL
LIN {X 0,Y 330.94,Z 736.933,A -85,B 0,C 180,E1 17583.123,E2 17583.123} C_VEL
LIN {X 0,Y 331.737,Z 715.447,A -85,B 0,C 180,E1 17583.659,E2 17583.659} C_VEL
LIN {X 0,Y 335.554,Z 572.427,A -85,B 0,C 180,E1 17586.656,E2 17586.656} C_VEL
LIN {X 0,Y 332.859,Z 542.143,A -85,B 0,C 180,E1 17587.683,E2 17587.683} C_VEL
LIN {X 0,Y 335.829,Z 525.242,A -85,B 0,C 180,E1 17589.813,E2 17589.813} C_VEL
LIN {X 0,Y 329.735,Z 505.78,A -85,B 0,C 180,E1 17593.429,E2 17593.429} C_VEL
LIN {X 0,Y 323.809,Z 488.669,A -85,B 0,C 180,E1 17596.968,E2 17596.968} C_VEL
LIN {X 0,Y 318.246,Z 474.017,A -85,B 0,C 180,E1 17600.374,E2 17600.374} C_VEL
LIN {X 0,Y 314.189,Z 463.821,A -85,B 0,C 180,E1 17603.04,E2 17603.04} C_VEL
LIN {X 0,Y 314.173,Z 463.645,A -85,B 0,C 180,E1 17607.498,E2 17607.498} C_VEL
LIN {X 0,Y 314.179,Z 463.643,A -85,B 0,C 180,E1 17611.901,E2 17611.901} C_VEL
LIN {X 0,Y 314.16,Z 463.659,A -85,B 0,C 180,E1 17616.435,E2 17616.435} C_VEL
LIN {X 0,Y 314.153,Z 463.665,A -85,B 0,C 180,E1 17620.956,E2 17620.956} C_VEL
LIN {X 0,Y 314.155,Z 463.631,A -85,B 0,C 180,E1 17625.438,E2 17625.438} C_VEL
LIN {X 0,Y 314.166,Z 463.646,A -85,B 0,C 180,E1 17629.919,E2 17629.919} C_VEL
LIN {X 0,Y 314.166,Z 463.649,A -85,B 0,C 180,E1 17634.338,E2 17634.338} C_VEL
LIN {X 0,Y 314.148,Z 463.629,A -85,B 0,C 180,E1 17638.724,E2 17638.724} C_VEL
LIN {X 0,Y 314.138,Z 463.657,A -85,B 0,C 180,E1 17643.102,E2 17643.102} C_VEL
LIN {X 0,Y 314.13,Z 463.625,A -85,B 0,C 180,E1 17647.499,E2 17647.499} C_VEL
LIN {X 0,Y 314.144,Z 463.659,A -85,B 0,C 180,E1 17651.94,E2 17651.94} C_VEL
LIN {X 0,Y 314.15,Z 463.622,A -85,B 0,C 180,E1 17656.265,E2 17656.265} C_VEL
LIN {X 0,Y 314.161,Z 463.655,A -85,B 0,C 180,E1 17660.688,E2 17660.688} C_VEL
LIN {X 0,Y 314.141,Z 463.626,A -85,B 0,C 180,E1 17665.045,E2 17665.045} C_VEL
LIN {X 0,Y 314.131,Z 463.663,A -85,B 0,C 180,E1 17669.352,E2 17669.352} C_VEL
LIN {X 0,Y 314.114,Z 463.628,A -85,B 0,C 180,E1 17673.819,E2 17673.819} C_VEL
LIN {X 0,Y 314.12,Z 463.669,A -85,B 0,C 180,E1 17678.166,E2 17678.166} C_VEL
LIN {X 0,Y 314.118,Z 463.64,A -85,B 0,C 180,E1 17682.44,E2 17682.44} C_VEL
LIN {X 0,Y 314.13,Z 463.643,A -85,B 0,C 180,E1 17686.816,E2 17686.816} C_VEL
LIN {X 0,Y 314.147,Z 463.661,A -85,B 0,C 180,E1 17691.241,E2 17691.241} C_VEL
LIN {X 0,Y 314.117,Z 463.67,A -85,B 0,C 180,E1 17695.708,E2 17695.708} C_VEL
LIN {X 0,Y 314.107,Z 463.671,A -85,B 0,C 180,E1 17700.016,E2 17700.016} C_VEL
LIN {X 0,Y 314.144,Z 463.941,A -85,B 0,C 180,E1 17702.412,E2 17702.412} C_VEL
LIN {X 0,Y 318.653,Z 476.701,A -85,B 0,C 180,E1 17706.123,E2 17706.123} C_VEL
LIN {X 0,Y 322.991,Z 490.319,A -85,B 0,C 180,E1 17709.716,E2 17709.716} C_VEL
LIN {X 0,Y 327.119,Z 505.083,A -85,B 0,C 180,E1 17713.302,E2 17713.302} C_VEL
LIN {X 0,Y 330.17,Z 517.661,A -85,B 0,C 180,E1 17716.158,E2 17716.158} C_VEL
LIN {X 0,Y 326.088,Z 544.164,A -85,B 0,C 180,E1 17720.825,E2 17720.825} C_VEL
LIN {X 0,Y 324.905,Z 553.165,A -85,B 0,C 180,E1 17722.334,E2 17722.334} C_VEL
LIN {X 0,Y 331.102,Z 593.183,A -85,B 0,C 180,E1 17723.895,E2 17723.895} C_VEL
LIN {X 0,Y 328.783,Z 666.9,A -85,B 0,C 180,E1 17725.549,E2 17725.549} C_VEL
LIN {X 0,Y 327.607,Z 674.564,A -85,B 0,C 180,E1 17725.645,E2 17725.645} C_VEL
LIN {X 0,Y 322.064,Z 691.556,A -85,B 0,C 180,E1 17725.765,E2 17725.765} C_VEL
LIN {X 0,Y 320.469,Z 697.944,A -85,B 0,C 180,E1 17725.949,E2 17725.949} C_VEL
LIN {X 0,Y 320.178,Z 701.139,A -85,B 0,C 180,E1 17726.111,E2 17726.111} C_VEL
LIN {X 0,Y 319.017,Z 715.625,A -85,B 0,C 180,E1 17727.035,E2 17727.035} C_VEL
LIN {X 0,Y 317.357,Z 730.872,A -85,B 0,C 180,E1 17728.375,E2 17728.375} C_VEL
LIN {X 0,Y 315.575,Z 744.232,A -85,B 0,C 180,E1 17729.909,E2 17729.909} C_VEL
LIN {X 0,Y 313.602,Z 757.235,A -85,B 0,C 180,E1 17731.827,E2 17731.827} C_VEL
LIN {X 0,Y 311.701,Z 768.543,A -85,B 0,C 180,E1 17733.955,E2 17733.955} C_VEL
LIN {X 0,Y 309.978,Z 778.371,A -85,B 0,C 180,E1 17736.296,E2 17736.296} C_VEL
LIN {X 0,Y 308.551,Z 786.403,A -85,B 0,C 180,E1 17738.76,E2 17738.76} C_VEL
LIN {X 0,Y 307.417,Z 793.081,A -85,B 0,C 180,E1 17741.443,E2 17741.443} C_VEL
LIN {X 0,Y 306.681,Z 797.95,A -85,B 0,C 180,E1 17744.153,E2 17744.153} C_VEL
LIN {X 0,Y 306.273,Z 801.554,A -85,B 0,C 180,E1 17747.282,E2 17747.282} C_VEL
LIN {X 0,Y 306.26,Z 803.111,A -85,B 0,C 180,E1 17750.246,E2 17750.246} C_VEL
LIN {X 0,Y 306.613,Z 802.983,A -85,B 0,C 180,E1 17753.239,E2 17753.239} C_VEL
LIN {X 0,Y 307.388,Z 801.051,A -85,B 0,C 180,E1 17756.255,E2 17756.255} C_VEL
LIN {X 0,Y 308.688,Z 797.229,A -85,B 0,C 180,E1 17759.281,E2 17759.281} C_VEL
LIN {X 0,Y 310.429,Z 791.681,A -85,B 0,C 180,E1 17762.103,E2 17762.103} C_VEL
LIN {X 0,Y 312.546,Z 784.655,A -85,B 0,C 180,E1 17764.711,E2 17764.711} C_VEL
LIN {X 0,Y 315.029,Z 775.788,A -85,B 0,C 180,E1 17767.189,E2 17767.189} C_VEL
LIN {X 0,Y 317.754,Z 765.314,A -85,B 0,C 180,E1 17769.466,E2 17769.466} C_VEL
LIN {X 0,Y 320.412,Z 753.772,A -85,B 0,C 180,E1 17771.418,E2 17771.418} C_VEL
LIN {X 0,Y 323.085,Z 740.745,A -85,B 0,C 180,E1 17773.152,E2 17773.152} C_VEL
LIN {X 0,Y 325.439,Z 726.661,A -85,B 0,C 180,E1 17774.59,E2 17774.59} C_VEL
LIN {X 0,Y 327.401,Z 711.894,A -85,B 0,C 180,E1 17775.737,E2 17775.737} C_VEL
LIN {X 0,Y 328.862,Z 695.722,A -85,B 0,C 180,E1 17776.621,E2 17776.621} C_VEL
LIN {X 0,Y 329.708,Z 679.451,A -85,B 0,C 180,E1 17777.184,E2 17777.184} C_VEL
LIN {X 0,Y 333.189,Z 595.772,A -85,B 0,C 180,E1 17779.17,E2 17779.17} C_VEL
LIN {X 0,Y 328.337,Z 567.954,A -85,B 0,C 180,E1 17780.682,E2 17780.682} C_VEL
LIN {X 0,Y 325.288,Z 553.106,A -85,B 0,C 180,E1 17781.618,E2 17781.618} C_VEL
LIN {X 0,Y 325.506,Z 550.516,A -85,B 0,C 180,E1 17781.988,E2 17781.988} C_VEL
LIN {X 0,Y 329.536,Z 531.171,A -85,B 0,C 180,E1 17785.617,E2 17785.617} C_VEL
LIN {X 0,Y 326.834,Z 519.157,A -85,B 0,C 180,E1 17788.935,E2 17788.935} C_VEL
LIN {X 0,Y 323.586,Z 507.758,A -85,B 0,C 180,E1 17792.475,E2 17792.475} C_VEL
LIN {X 0,Y 320.42,Z 498.207,A -85,B 0,C 180,E1 17795.871,E2 17795.871} C_VEL
LIN {X 0,Y 317.133,Z 489.207,A -85,B 0,C 180,E1 17799.515,E2 17799.515} C_VEL
LIN {X 0,Y 313.962,Z 481.593,A -85,B 0,C 180,E1 17803.153,E2 17803.153} C_VEL
LIN {X 0,Y 312.02,Z 477.308,A -85,B 0,C 180,E1 17805.525,E2 17805.525} C_VEL
LIN {X 0,Y 310.291,Z 473.404,A -85,B 0,C 180,E1 17807.909,E2 17807.909} C_VEL
LIN {X 0,Y 308.086,Z 468.848,A -85,B 0,C 180,E1 17811.226,E2 17811.226} C_VEL
LIN {X 0,Y 306.242,Z 464.736,A -85,B 0,C 180,E1 17815.13,E2 17815.13} C_VEL
LIN {X 0,Y 306.235,Z 464.621,A -85,B 0,C 180,E1 17819.625,E2 17819.625} C_VEL
LIN {X 0,Y 306.226,Z 464.622,A -85,B 0,C 180,E1 17824.119,E2 17824.119} C_VEL
LIN {X 0,Y 306.224,Z 464.627,A -85,B 0,C 180,E1 17828.638,E2 17828.638} C_VEL
LIN {X 0,Y 306.229,Z 464.631,A -85,B 0,C 180,E1 17833.212,E2 17833.212} C_VEL
LIN {X 0,Y 306.232,Z 464.638,A -85,B 0,C 180,E1 17837.677,E2 17837.677} C_VEL
LIN {X 0,Y 306.284,Z 464.971,A -85,B 0,C 180,E1 17840.344,E2 17840.344} C_VEL
LIN {X 0,Y 308.985,Z 470.425,A -85,B 0,C 180,E1 17844.877,E2 17844.877} C_VEL
LIN {X 0,Y 311.456,Z 475.298,A -85,B 0,C 180,E1 17848.016,E2 17848.016} C_VEL
LIN {X 0,Y 313.661,Z 479.759,A -85,B 0,C 180,E1 17850.454,E2 17850.454} C_VEL
LIN {X 0,Y 315.918,Z 484.631,A -85,B 0,C 180,E1 17852.765,E2 17852.765} C_VEL
LIN {X 0,Y 317.965,Z 489.117,A -85,B 0,C 180,E1 17854.692,E2 17854.692} C_VEL
LIN {X 0,Y 321.122,Z 496.15,A -85,B 0,C 180,E1 17857.384,E2 17857.384} C_VEL
LIN {X 0,Y 325.246,Z 506.109,A -85,B 0,C 180,E1 17860.671,E2 17860.671} C_VEL
LIN {X 0,Y 329.662,Z 518.097,A -85,B 0,C 180,E1 17864.044,E2 17864.044} C_VEL
LIN {X 0,Y 333.804,Z 531.177,A -85,B 0,C 180,E1 17867.211,E2 17867.211} C_VEL
LIN {X 0,Y 335.149,Z 536.18,A -85,B 0,C 180,E1 17868.296,E2 17868.296} C_VEL
LIN {X 0,Y 333.418,Z 544.139,A -85,B 0,C 180,E1 17869.308,E2 17869.308} C_VEL
LIN {X 0,Y 336.448,Z 574.614,A -85,B 0,C 180,E1 17870.611,E2 17870.611} C_VEL
LIN {X 0,Y 335.603,Z 599.864,A -85,B 0,C 180,E1 17871.192,E2 17871.192} C_VEL
LIN {X 0,Y 330.674,Z 730.107,A -85,B 0,C 180,E1 17874.037,E2 17874.037} C_VEL
LIN {X 0,Y 329.017,Z 748.356,A -85,B 0,C 180,E1 17874.713,E2 17874.713} C_VEL
LIN {X 0,Y 326.547,Z 766.632,A -85,B 0,C 180,E1 17875.71,E2 17875.71} C_VEL
LIN {X 0,Y 323.724,Z 783.461,A -85,B 0,C 180,E1 17876.966,E2 17876.966} C_VEL
LIN {X 0,Y 320.642,Z 799.442,A -85,B 0,C 180,E1 17878.513,E2 17878.513} C_VEL
LIN {X 0,Y 317.408,Z 814.805,A -85,B 0,C 180,E1 17880.391,E2 17880.391} C_VEL
LIN {X 0,Y 314.061,Z 829.589,A -85,B 0,C 180,E1 17882.652,E2 17882.652} C_VEL
LIN {X 0,Y 311.161,Z 842.585,A -85,B 0,C 180,E1 17885.106,E2 17885.106} C_VEL
LIN {X 0,Y 308.551,Z 854.812,A -85,B 0,C 180,E1 17887.938,E2 17887.938} C_VEL
LIN {X 0,Y 306.545,Z 865.729,A -85,B 0,C 180,E1 17891.066,E2 17891.066} C_VEL
LIN {X 0,Y 305.284,Z 874.85,A -85,B 0,C 180,E1 17894.344,E2 17894.344} C_VEL
LIN {X 0,Y 304.778,Z 882.095,A -85,B 0,C 180,E1 17897.688,E2 17897.688} C_VEL
LIN {X 0,Y 304.87,Z 887.599,A -85,B 0,C 180,E1 17901.133,E2 17901.133} C_VEL
LIN {X 0,Y 305.321,Z 891.088,A -85,B 0,C 180,E1 17904.362,E2 17904.362} C_VEL
LIN {X 0,Y 305.754,Z 892.862,A -85,B 0,C 180,E1 17907.376,E2 17907.376} C_VEL
LIN {X 0,Y 305.94,Z 893.117,A -85,B 0,C 180,E1 17910.375,E2 17910.375} C_VEL
LIN {X 0,Y 305.763,Z 891.859,A -85,B 0,C 180,E1 17913.375,E2 17913.375} C_VEL
LIN {X 0,Y 305.352,Z 889.063,A -85,B 0,C 180,E1 17916.392,E2 17916.392} C_VEL
LIN {X 0,Y 304.995,Z 884.365,A -85,B 0,C 180,E1 17919.625,E2 17919.625} C_VEL
LIN {X 0,Y 304.986,Z 877.796,A -85,B 0,C 180,E1 17922.882,E2 17922.882} C_VEL
LIN {X 0,Y 305.474,Z 869.746,A -85,B 0,C 180,E1 17925.959,E2 17925.959} C_VEL
LIN {X 0,Y 306.581,Z 859.651,A -85,B 0,C 180,E1 17929.035,E2 17929.035} C_VEL
LIN {X 0,Y 308.259,Z 847.945,A -85,B 0,C 180,E1 17931.902,E2 17931.902} C_VEL
LIN {X 0,Y 310.339,Z 835.102,A -85,B 0,C 180,E1 17934.457,E2 17934.457} C_VEL
LIN {X 0,Y 312.749,Z 820.685,A -85,B 0,C 180,E1 17936.794,E2 17936.794} C_VEL
LIN {X 0,Y 315.321,Z 805.243,A -85,B 0,C 180,E1 17938.815,E2 17938.815} C_VEL
LIN {X 0,Y 317.717,Z 789.725,A -85,B 0,C 180,E1 17940.443,E2 17940.443} C_VEL
LIN {X 0,Y 319.994,Z 773.269,A -85,B 0,C 180,E1 17941.8,E2 17941.8} C_VEL
LIN {X 0,Y 322.083,Z 755.406,A -85,B 0,C 180,E1 17942.906,E2 17942.906} C_VEL
LIN {X 0,Y 323.633,Z 736.924,A -85,B 0,C 180,E1 17943.694,E2 17943.694} C_VEL
LIN {X 0,Y 324.452,Z 716.389,A -85,B 0,C 180,E1 17944.228,E2 17944.228} C_VEL
LIN {X 0,Y 328.433,Z 573.174,A -85,B 0,C 180,E1 17947.281,E2 17947.281} C_VEL
LIN {X 0,Y 325.732,Z 542.662,A -85,B 0,C 180,E1 17948.32,E2 17948.32} C_VEL
LIN {X 0,Y 328.358,Z 527.411,A -85,B 0,C 180,E1 17950.277,E2 17950.277} C_VEL
LIN {X 0,Y 322.359,Z 508.081,A -85,B 0,C 180,E1 17953.979,E2 17953.979} C_VEL
LIN {X 0,Y 316.686,Z 491.603,A -85,B 0,C 180,E1 17957.495,E2 17957.495} C_VEL
LIN {X 0,Y 310.597,Z 475.558,A -85,B 0,C 180,E1 17961.354,E2 17961.354} C_VEL
LIN {X 0,Y 306.244,Z 464.801,A -85,B 0,C 180,E1 17964.315,E2 17964.315} C_VEL
LIN {X 0,Y 306.223,Z 464.635,A -85,B 0,C 180,E1 17968.943,E2 17968.943} C_VEL
LIN {X 0,Y 306.231,Z 464.627,A -85,B 0,C 180,E1 17973.461,E2 17973.461} C_VEL
LIN {X 0,Y 306.238,Z 464.621,A -85,B 0,C 180,E1 17978.011,E2 17978.011} C_VEL
LIN {X 0,Y 306.218,Z 464.646,A -85,B 0,C 180,E1 17982.519,E2 17982.519} C_VEL
LIN {X 0,Y 306.209,Z 464.642,A -85,B 0,C 180,E1 17986.98,E2 17986.98} C_VEL
LIN {X 0,Y 306.212,Z 464.613,A -85,B 0,C 180,E1 17991.551,E2 17991.551} C_VEL
LIN {X 0,Y 306.226,Z 464.654,A -85,B 0,C 180,E1 17996.069,E2 17996.069} C_VEL
LIN {X 0,Y 306.216,Z 464.605,A -85,B 0,C 180,E1 18000.562,E2 18000.562} C_VEL
LIN {X 0,Y 306.2,Z 464.65,A -85,B 0,C 180,E1 18005.16,E2 18005.16} C_VEL
LIN {X 0,Y 306.197,Z 464.609,A -85,B 0,C 180,E1 18009.777,E2 18009.777} C_VEL
LIN {X 0,Y 306.228,Z 464.643,A -85,B 0,C 180,E1 18014.368,E2 18014.368} C_VEL
LIN {X 0,Y 306.207,Z 464.61,A -85,B 0,C 180,E1 18018.861,E2 18018.861} C_VEL
LIN {X 0,Y 306.194,Z 464.648,A -85,B 0,C 180,E1 18023.274,E2 18023.274} C_VEL
LIN {X 0,Y 306.183,Z 464.624,A -85,B 0,C 180,E1 18027.839,E2 18027.839} C_VEL
LIN {X 0,Y 306.189,Z 464.635,A -85,B 0,C 180,E1 18032.245,E2 18032.245} C_VEL
LIN {X 0,Y 306.203,Z 464.646,A -85,B 0,C 180,E1 18036.696,E2 18036.696} C_VEL
LIN {X 0,Y 306.214,Z 464.618,A -85,B 0,C 180,E1 18041.038,E2 18041.038} C_VEL
LIN {X 0,Y 306.18,Z 464.651,A -85,B 0,C 180,E1 18045.666,E2 18045.666} C_VEL
LIN {X 0,Y 306.169,Z 464.661,A -85,B 0,C 180,E1 18050.202,E2 18050.202} C_VEL
LIN {X 0,Y 306.176,Z 464.649,A -85,B 0,C 180,E1 18054.728,E2 18054.728} C_VEL
LIN {X 0,Y 306.197,Z 464.648,A -85,B 0,C 180,E1 18059.183,E2 18059.183} C_VEL
LIN {X 0,Y 306.224,Z 464.868,A -85,B 0,C 180,E1 18061.156,E2 18061.156} C_VEL
LIN {X 0,Y 310.841,Z 477.842,A -85,B 0,C 180,E1 18065.107,E2 18065.107} C_VEL
LIN {X 0,Y 315.209,Z 491.455,A -85,B 0,C 180,E1 18068.843,E2 18068.843} C_VEL
LIN {X 0,Y 319.483,Z 506.64,A -85,B 0,C 180,E1 18072.658,E2 18072.658} C_VEL
LIN {X 0,Y 322.727,Z 520.312,A -85,B 0,C 180,E1 18075.832,E2 18075.832} C_VEL
LIN {X 0,Y 318.453,Z 546.915,A -85,B 0,C 180,E1 18080.603,E2 18080.603} C_VEL
LIN {X 0,Y 317.645,Z 553.019,A -85,B 0,C 180,E1 18081.623,E2 18081.623} C_VEL
LIN {X 0,Y 323.945,Z 594.162,A -85,B 0,C 180,E1 18083.279,E2 18083.279} C_VEL
LIN {X 0,Y 321.012,Z 685.362,A -85,B 0,C 180,E1 18085.422,E2 18085.422} C_VEL
LIN {X 0,Y 320.178,Z 701.139,A -85,B 0,C 180,E1 18086.111,E2 18086.111} C_VEL
LIN {X 0,Y 318.739,Z 708.525,A -85,B 0,C 180,E1 18086.462,E2 18086.462} C_VEL
LIN {X 0,Y 313.042,Z 722.618,A -85,B 0,C 180,E1 18087.146,E2 18087.146} C_VEL
LIN {X 0,Y 310.298,Z 730.457,A -85,B 0,C 180,E1 18087.73,E2 18087.73} C_VEL
LIN {X 0,Y 309.742,Z 733.349,A -85,B 0,C 180,E1 18088.015,E2 18088.015} C_VEL
LIN {X 0,Y 307.745,Z 747.315,A -85,B 0,C 180,E1 18089.72,E2 18089.72} C_VEL
LIN {X 0,Y 305.82,Z 759.363,A -85,B 0,C 180,E1 18091.592,E2 18091.592} C_VEL
LIN {X 0,Y 303.864,Z 770.429,A -85,B 0,C 180,E1 18093.773,E2 18093.773} C_VEL
LIN {X 0,Y 302.162,Z 779.749,A -85,B 0,C 180,E1 18096.078,E2 18096.078} C_VEL
LIN {X 0,Y 300.585,Z 788.248,A -85,B 0,C 180,E1 18098.801,E2 18098.801} C_VEL
LIN {X 0,Y 299.446,Z 794.758,A -85,B 0,C 180,E1 18101.557,E2 18101.557} C_VEL
LIN {X 0,Y 298.662,Z 799.868,A -85,B 0,C 180,E1 18104.642,E2 18104.642} C_VEL
LIN {X 0,Y 298.336,Z 802.917,A -85,B 0,C 180,E1 18107.555,E2 18107.555} C_VEL
LIN {X 0,Y 298.382,Z 804.382,A -85,B 0,C 180,E1 18110.805,E2 18110.805} C_VEL
LIN {X 0,Y 298.832,Z 804.009,A -85,B 0,C 180,E1 18113.882,E2 18113.882} C_VEL
LIN {X 0,Y 299.829,Z 801.633,A -85,B 0,C 180,E1 18117.185,E2 18117.185} C_VEL
LIN {X 0,Y 301.225,Z 797.721,A -85,B 0,C 180,E1 18120.08,E2 18120.08} C_VEL
LIN {X 0,Y 303.172,Z 791.934,A -85,B 0,C 180,E1 18122.968,E2 18122.968} C_VEL
LIN {X 0,Y 305.493,Z 784.586,A -85,B 0,C 180,E1 18125.632,E2 18125.632} C_VEL
LIN {X 0,Y 308.099,Z 775.786,A -85,B 0,C 180,E1 18128.068,E2 18128.068} C_VEL
LIN {X 0,Y 310.869,Z 765.605,A -85,B 0,C 180,E1 18130.277,E2 18130.277} C_VEL
LIN {X 0,Y 313.824,Z 753.433,A -85,B 0,C 180,E1 18132.339,E2 18132.339} C_VEL
LIN {X 0,Y 316.53,Z 740.713,A -85,B 0,C 180,E1 18134.022,E2 18134.022} C_VEL
LIN {X 0,Y 318.995,Z 726.596,A -85,B 0,C 180,E1 18135.467,E2 18135.467} C_VEL
LIN {X 0,Y 320.989,Z 711.991,A -85,B 0,C 180,E1 18136.598,E2 18136.598} C_VEL
LIN {X 0,Y 322.543,Z 695.369,A -85,B 0,C 180,E1 18137.505,E2 18137.505} C_VEL
LIN {X 0,Y 323.412,Z 678.61,A -85,B 0,C 180,E1 18138.069,E2 18138.069} C_VEL
LIN {X 0,Y 326.984,Z 597.139,A -85,B 0,C 180,E1 18140.027,E2 18140.027} C_VEL
LIN {X 0,Y 322.153,Z 569.003,A -85,B 0,C 180,E1 18141.615,E2 18141.615} C_VEL
LIN {X 0,Y 318.923,Z 553.111,A -85,B 0,C 180,E1 18142.652,E2 18142.652} C_VEL
LIN {X 0,Y 318.993,Z 551.059,A -85,B 0,C 180,E1 18142.912,E2 18142.912} C_VEL
LIN {X 0,Y 322.647,Z 534.431,A -85,B 0,C 180,E1 18146.095,E2 18146.095} C_VEL
LIN {X 0,Y 320.095,Z 522.804,A -85,B 0,C 180,E1 18149.392,E2 18149.392} C_VEL
LIN {X 0,Y 317.003,Z 511.622,A -85,B 0,C 180,E1 18152.987,E2 18152.987} C_VEL
LIN {X 0,Y 313.771,Z 501.817,A -85,B 0,C 180,E1 18156.597,E2 18156.597} C_VEL
LIN {X 0,Y 310.752,Z 493.672,A -85,B 0,C 180,E1 18160.058,E2 18160.058} C_VEL
LIN {X 0,Y 308.052,Z 486.868,A -85,B 0,C 180,E1 18163.403,E2 18163.403} C_VEL
LIN {X 0,Y 306.156,Z 482.619,A -85,B 0,C 180,E1 18165.821,E2 18165.821} C_VEL
LIN {X 0,Y 304.646,Z 479.035,A -85,B 0,C 180,E1 18168.067,E2 18168.067} C_VEL
LIN {X 0,Y 302.498,Z 474.518,A -85,B 0,C 180,E1 18171.446,E2 18171.446} C_VEL
LIN {X 0,Y 300.416,Z 470.159,A -85,B 0,C 180,E1 18175.609,E2 18175.609} C_VEL
LIN {X 0,Y 298.32,Z 465.888,A -85,B 0,C 180,E1 18182.497,E2 18182.497} C_VEL
LIN {X 0,Y 298.296,Z 465.657,A -85,B 0,C 180,E1 18187.124,E2 18187.124} C_VEL
LIN {X 0,Y 298.309,Z 465.756,A -85,B 0,C 180,E1 18191.797,E2 18191.797} C_VEL
LIN {X 0,Y 298.748,Z 467.451,A -85,B 0,C 180,E1 18195.331,E2 18195.331} C_VEL
LIN {X 0,Y 301.067,Z 471.209,A -85,B 0,C 180,E1 18200.408,E2 18200.408} C_VEL
LIN {X 0,Y 303.67,Z 476.365,A -85,B 0,C 180,E1 18204.718,E2 18204.718} C_VEL
LIN {X 0,Y 306.038,Z 481.157,A -85,B 0,C 180,E1 18207.852,E2 18207.852} C_VEL
LIN {X 0,Y 308.235,Z 485.788,A -85,B 0,C 180,E1 18210.4,E2 18210.4} C_VEL
LIN {X 0,Y 310.311,Z 490.228,A -85,B 0,C 180,E1 18212.554,E2 18212.554} C_VEL
LIN {X 0,Y 313.465,Z 497.028,A -85,B 0,C 180,E1 18215.487,E2 18215.487} C_VEL
LIN {X 0,Y 317.893,Z 507.715,A -85,B 0,C 180,E1 18219.31,E2 18219.31} C_VEL
LIN {X 0,Y 322.406,Z 519.854,A -85,B 0,C 180,E1 18222.955,E2 18222.955} C_VEL
LIN {X 0,Y 326.552,Z 532.821,A -85,B 0,C 180,E1 18226.269,E2 18226.269} C_VEL
LIN {X 0,Y 328.278,Z 539.314,A -85,B 0,C 180,E1 18227.742,E2 18227.742} C_VEL
LIN {X 0,Y 327.215,Z 544.38,A -85,B 0,C 180,E1 18228.373,E2 18228.373} C_VEL
LIN {X 0,Y 330.243,Z 575.401,A -85,B 0,C 180,E1 18229.744,E2 18229.744} C_VEL
LIN {X 0,Y 329.873,Z 588.966,A -85,B 0,C 180,E1 18230.077,E2 18230.077} C_VEL
LIN {X 0,Y 324.217,Z 729.35,A -85,B 0,C 180,E1 18233.198,E2 18233.198} C_VEL
LIN {X 0,Y 322.498,Z 747.541,A -85,B 0,C 180,E1 18233.882,E2 18233.882} C_VEL
LIN {X 0,Y 319.906,Z 765.863,A -85,B 0,C 180,E1 18234.895,E2 18234.895} C_VEL
LIN {X 0,Y 316.947,Z 782.783,A -85,B 0,C 180,E1 18236.177,E2 18236.177} C_VEL
LIN {X 0,Y 313.734,Z 798.647,A -85,B 0,C 180,E1 18237.738,E2 18237.738} C_VEL
LIN {X 0,Y 310.382,Z 813.769,A -85,B 0,C 180,E1 18239.619,E2 18239.619} C_VEL
LIN {X 0,Y 306.858,Z 828.505,A -85,B 0,C 180,E1 18241.912,E2 18241.912} C_VEL
LIN {X 0,Y 303.729,Z 841.681,A -85,B 0,C 180,E1 18244.454,E2 18244.454} C_VEL
LIN {X 0,Y 300.957,Z 853.794,A -85,B 0,C 180,E1 18247.333,E2 18247.333} C_VEL
LIN {X 0,Y 298.829,Z 864.4,A -85,B 0,C 180,E1 18250.453,E2 18250.453} C_VEL
LIN {X 0,Y 297.428,Z 873.509,A -85,B 0,C 180,E1 18253.799,E2 18253.799} C_VEL
LIN {X 0,Y 296.81,Z 881.013,A -85,B 0,C 180,E1 18257.352,E2 18257.352} C_VEL
LIN {X 0,Y 296.881,Z 886.489,A -85,B 0,C 180,E1 18260.893,E2 18260.893} C_VEL
LIN {X 0,Y 297.349,Z 889.951,A -85,B 0,C 180,E1 18264.211,E2 18264.211} C_VEL
LIN {X 0,Y 297.822,Z 891.71,A -85,B 0,C 180,E1 18267.306,E2 18267.306} C_VEL
LIN {X 0,Y 298.028,Z 891.93,A -85,B 0,C 180,E1 18270.385,E2 18270.385} C_VEL
LIN {X 0,Y 297.834,Z 890.616,A -85,B 0,C 180,E1 18273.465,E2 18273.465} C_VEL
LIN {X 0,Y 297.391,Z 887.75,A -85,B 0,C 180,E1 18276.564,E2 18276.564} C_VEL
LIN {X 0,Y 297.023,Z 882.972,A -85,B 0,C 180,E1 18279.886,E2 18279.886} C_VEL
LIN {X 0,Y 297.038,Z 876.314,A -85,B 0,C 180,E1 18283.232,E2 18283.232} C_VEL
LIN {X 0,Y 297.595,Z 868.165,A -85,B 0,C 180,E1 18286.393,E2 18286.393} C_VEL
LIN {X 0,Y 298.801,Z 857.938,A -85,B 0,C 180,E1 18289.55,E2 18289.55} C_VEL
LIN {X 0,Y 300.608,Z 846.043,A -85,B 0,C 180,E1 18292.489,E2 18292.489} C_VEL
LIN {X 0,Y 302.81,Z 833.067,A -85,B 0,C 180,E1 18295.098,E2 18295.098} C_VEL
LIN {X 0,Y 305.396,Z 818.395,A -85,B 0,C 180,E1 18297.493,E2 18297.493} C_VEL
LIN {X 0,Y 307.97,Z 803.407,A -85,B 0,C 180,E1 18299.463,E2 18299.463} C_VEL
LIN {X 0,Y 310.482,Z 787.638,A -85,B 0,C 180,E1 18301.123,E2 18301.123} C_VEL
LIN {X 0,Y 312.811,Z 771.158,A -85,B 0,C 180,E1 18302.479,E2 18302.479} C_VEL
LIN {X 0,Y 314.933,Z 753.174,A -85,B 0,C 180,E1 18303.575,E2 18303.575} C_VEL
LIN {X 0,Y 316.437,Z 734.941,A -85,B 0,C 180,E1 18304.341,E2 18304.341} C_VEL
LIN {X 0,Y 317.336,Z 711.098,A -85,B 0,C 180,E1 18304.94,E2 18304.94} C_VEL
LIN {X 0,Y 321.331,Z 573.915,A -85,B 0,C 180,E1 18307.927,E2 18307.927} C_VEL
LIN {X 0,Y 318.677,Z 542.554,A -85,B 0,C 180,E1 18309.034,E2 18309.034} C_VEL
LIN {X 0,Y 320.989,Z 529.869,A -85,B 0,C 180,E1 18310.712,E2 18310.712} C_VEL
LIN {X 0,Y 315.134,Z 510.852,A -85,B 0,C 180,E1 18314.449,E2 18314.449} C_VEL
LIN {X 0,Y 309.552,Z 494.539,A -85,B 0,C 180,E1 18318.04,E2 18318.04} C_VEL
LIN {X 0,Y 304.141,Z 480.149,A -85,B 0,C 180,E1 18321.587,E2 18321.587} C_VEL
LIN {X 0,Y 299.455,Z 468.91,A -85,B 0,C 180,E1 18324.716,E2 18324.716} C_VEL
LIN {X 0,Y 298.314,Z 465.763,A -85,B 0,C 180,E1 18325.731,E2 18325.731} C_VEL
LIN {X 0,Y 298.289,Z 465.642,A -85,B 0,C 180,E1 18330.258,E2 18330.258} C_VEL
LIN {X 0,Y 298.278,Z 465.635,A -85,B 0,C 180,E1 18334.833,E2 18334.833} C_VEL
LIN {X 0,Y 298.284,Z 465.615,A -85,B 0,C 180,E1 18339.393,E2 18339.393} C_VEL
LIN {X 0,Y 298.294,Z 465.608,A -85,B 0,C 180,E1 18343.847,E2 18343.847} C_VEL
LIN {X 0,Y 298.285,Z 465.644,A -85,B 0,C 180,E1 18348.398,E2 18348.398} C_VEL
LIN {X 0,Y 298.264,Z 465.606,A -85,B 0,C 180,E1 18353.069,E2 18353.069} C_VEL
LIN {X 0,Y 298.273,Z 465.623,A -85,B 0,C 180,E1 18357.695,E2 18357.695} C_VEL
LIN {X 0,Y 298.282,Z 465.612,A -85,B 0,C 180,E1 18362.114,E2 18362.114} C_VEL
LIN {X 0,Y 298.285,Z 465.613,A -85,B 0,C 180,E1 18366.545,E2 18366.545} C_VEL
LIN {X 0,Y 298.261,Z 465.619,A -85,B 0,C 180,E1 18371.016,E2 18371.016} C_VEL
LIN {X 0,Y 298.25,Z 465.613,A -85,B 0,C 180,E1 18375.557,E2 18375.557} C_VEL
LIN {X 0,Y 298.266,Z 465.626,A -85,B 0,C 180,E1 18380.199,E2 18380.199} C_VEL
LIN {X 0,Y 298.275,Z 465.604,A -85,B 0,C 180,E1 18384.71,E2 18384.71} C_VEL
LIN {X 0,Y 298.255,Z 465.638,A -85,B 0,C 180,E1 18389.305,E2 18389.305} C_VEL
LIN {X 0,Y 298.237,Z 465.603,A -85,B 0,C 180,E1 18393.816,E2 18393.816} C_VEL
LIN {X 0,Y 298.248,Z 465.647,A -85,B 0,C 180,E1 18398.331,E2 18398.331} C_VEL
LIN {X 0,Y 298.26,Z 465.62,A -85,B 0,C 180,E1 18402.885,E2 18402.885} C_VEL
LIN {X 0,Y 298.251,Z 465.615,A -85,B 0,C 180,E1 18407.375,E2 18407.375} C_VEL
LIN {X 0,Y 298.23,Z 465.631,A -85,B 0,C 180,E1 18411.91,E2 18411.91} C_VEL
LIN {X 0,Y 298.229,Z 465.635,A -85,B 0,C 180,E1 18416.597,E2 18416.597} C_VEL
LIN {X 0,Y 298.273,Z 465.919,A -85,B 0,C 180,E1 18419.867,E2 18419.867} C_VEL
LIN {X 0,Y 302.884,Z 478.494,A -85,B 0,C 180,E1 18423.886,E2 18423.886} C_VEL
LIN {X 0,Y 307.26,Z 491.838,A -85,B 0,C 180,E1 18427.721,E2 18427.721} C_VEL
LIN {X 0,Y 311.419,Z 506.532,A -85,B 0,C 180,E1 18431.563,E2 18431.563} C_VEL
LIN {X 0,Y 315.242,Z 522.187,A -85,B 0,C 180,E1 18435.326,E2 18435.326} C_VEL
LIN {X 0,Y 312.418,Z 539.745,A -85,B 0,C 180,E1 18438.555,E2 18438.555} C_VEL
LIN {X 0,Y 310.429,Z 552.834,A -85,B 0,C 180,E1 18440.878,E2 18440.878} C_VEL
LIN {X 0,Y 316.815,Z 595.338,A -85,B 0,C 180,E1 18442.642,E2 18442.642} C_VEL
LIN {X 0,Y 313.772,Z 685.982,A -85,B 0,C 180,E1 18444.816,E2 18444.816} C_VEL
LIN {X 0,Y 312.806,Z 703.267,A -85,B 0,C 180,E1 18445.6,E2 18445.6} C_VEL
LIN {X 0,Y 311.506,Z 718.057,A -85,B 0,C 180,E1 18446.606,E2 18446.606} C_VEL
LIN {X 0,Y 309.803,Z 732.88,A -85,B 0,C 180,E1 18447.965,E2 18447.965} C_VEL
LIN {X 0,Y 309.742,Z 733.349,A -85,B 0,C 180,E1 18448.015,E2 18448.015} C_VEL
LIN {X 0,Y 307.935,Z 739.985,A -85,B 0,C 180,E1 18448.688,E2 18448.688} C_VEL
LIN {X 0,Y 301.623,Z 752.481,A -85,B 0,C 180,E1 18450.01,E2 18450.01} C_VEL
LIN {X 0,Y 298.625,Z 759.217,A -85,B 0,C 180,E1 18450.961,E2 18450.961} C_VEL
LIN {X 0,Y 298.003,Z 761.625,A -85,B 0,C 180,E1 18451.383,E2 18451.383} C_VEL
LIN {X 0,Y 295.955,Z 772.751,A -85,B 0,C 180,E1 18453.68,E2 18453.68} C_VEL
LIN {X 0,Y 294.082,Z 782.433,A -85,B 0,C 180,E1 18456.246,E2 18456.246} C_VEL
LIN {X 0,Y 292.524,Z 790.617,A -85,B 0,C 180,E1 18459.046,E2 18459.046} C_VEL
LIN {X 0,Y 291.342,Z 797.139,A -85,B 0,C 180,E1 18462.084,E2 18462.084} C_VEL
LIN {X 0,Y 290.652,Z 801.738,A -85,B 0,C 180,E1 18465.155,E2 18465.155} C_VEL
LIN {X 0,Y 290.384,Z 804.655,A -85,B 0,C 180,E1 18468.468,E2 18468.468} C_VEL
LIN {X 0,Y 290.545,Z 805.631,A -85,B 0,C 180,E1 18471.606,E2 18471.606} C_VEL
LIN {X 0,Y 291.194,Z 804.792,A -85,B 0,C 180,E1 18474.982,E2 18474.982} C_VEL
LIN {X 0,Y 292.284,Z 802.244,A -85,B 0,C 180,E1 18478.044,E2 18478.044} C_VEL
LIN {X 0,Y 293.96,Z 797.838,A -85,B 0,C 180,E1 18481.131,E2 18481.131} C_VEL
LIN {X 0,Y 295.988,Z 792.156,A -85,B 0,C 180,E1 18483.874,E2 18483.874} C_VEL
LIN {X 0,Y 298.535,Z 784.526,A -85,B 0,C 180,E1 18486.595,E2 18486.595} C_VEL
LIN {X 0,Y 301.372,Z 775.466,A -85,B 0,C 180,E1 18489.076,E2 18489.076} C_VEL
LIN {X 0,Y 304.492,Z 764.348,A -85,B 0,C 180,E1 18491.427,E2 18491.427} C_VEL
LIN {X 0,Y 307.399,Z 752.856,A -85,B 0,C 180,E1 18493.338,E2 18493.338} C_VEL
LIN {X 0,Y 310.417,Z 738.882,A -85,B 0,C 180,E1 18495.137,E2 18495.137} C_VEL
LIN {X 0,Y 312.86,Z 725.103,A -85,B 0,C 180,E1 18496.507,E2 18496.507} C_VEL
LIN {X 0,Y 314.922,Z 709.753,A -85,B 0,C 180,E1 18497.643,E2 18497.643} C_VEL
LIN {X 0,Y 316.369,Z 694.013,A -85,B 0,C 180,E1 18498.464,E2 18498.464} C_VEL
LIN {X 0,Y 317.387,Z 673.501,A -85,B 0,C 180,E1 18499.097,E2 18499.097} C_VEL
LIN {X 0,Y 320.855,Z 598.513,A -85,B 0,C 180,E1 18500.918,E2 18500.918} C_VEL
LIN {X 0,Y 316.108,Z 570.269,A -85,B 0,C 180,E1 18502.574,E2 18502.574} C_VEL
LIN {X 0,Y 312.583,Z 552.086,A -85,B 0,C 180,E1 18503.831,E2 18503.831} C_VEL
LIN {X 0,Y 315.8,Z 537.787,A -85,B 0,C 180,E1 18506.57,E2 18506.57} C_VEL
LIN {X 0,Y 313.354,Z 526.292,A -85,B 0,C 180,E1 18509.936,E2 18509.936} C_VEL
LIN {X 0,Y 310.344,Z 515.288,A -85,B 0,C 180,E1 18513.601,E2 18513.601} C_VEL
LIN {X 0,Y 307.306,Z 505.776,A -85,B 0,C 180,E1 18517.22,E2 18517.22} C_VEL
LIN {X 0,Y 303.954,Z 496.457,A -85,B 0,C 180,E1 18521.392,E2 18521.392} C_VEL
LIN {X 0,Y 300.998,Z 489.027,A -85,B 0,C 180,E1 18525.377,E2 18525.377} C_VEL
LIN {X 0,Y 298.853,Z 484.446,A -85,B 0,C 180,E1 18528.419,E2 18528.419} C_VEL
LIN {X 0,Y 297.073,Z 480.396,A -85,B 0,C 180,E1 18531.483,E2 18531.483} C_VEL
LIN {X 0,Y 295.043,Z 476.069,A -85,B 0,C 180,E1 18535.724,E2 18535.724} C_VEL
LIN {X 0,Y 293.026,Z 471.836,A -85,B 0,C 180,E1 18542.738,E2 18542.738} C_VEL
LIN {X 0,Y 292.513,Z 471.176,A -85,B 0,C 180,E1 18547.66,E2 18547.66} C_VEL
LIN {X 0,Y 293.115,Z 471.937,A -85,B 0,C 180,E1 18552.409,E2 18552.409} C_VEL
LIN {X 0,Y 295.766,Z 476.896,A -85,B 0,C 180,E1 18559.983,E2 18559.983} C_VEL
LIN {X 0,Y 298.351,Z 482.298,A -85,B 0,C 180,E1 18564.554,E2 18564.554} C_VEL
LIN {X 0,Y 300.543,Z 486.738,A -85,B 0,C 180,E1 18567.544,E2 18567.544} C_VEL
LIN {X 0,Y 302.671,Z 491.367,A -85,B 0,C 180,E1 18570.14,E2 18570.14} C_VEL
LIN {X 0,Y 304.912,Z 496.357,A -85,B 0,C 180,E1 18572.569,E2 18572.569} C_VEL
LIN {X 0,Y 307.85,Z 502.853,A -85,B 0,C 180,E1 18575.392,E2 18575.392} C_VEL
LIN {X 0,Y 312.068,Z 513.25,A -85,B 0,C 180,E1 18579.162,E2 18579.162} C_VEL
LIN {X 0,Y 316.13,Z 524.416,A -85,B 0,C 180,E1 18582.597,E2 18582.597} C_VEL
LIN {X 0,Y 320.104,Z 537.138,A -85,B 0,C 180,E1 18585.923,E2 18585.923} C_VEL
LIN {X 0,Y 321.406,Z 542.555,A -85,B 0,C 180,E1 18587.178,E2 18587.178} C_VEL
LIN {X 0,Y 321.154,Z 545.1,A -85,B 0,C 180,E1 18587.425,E2 18587.425} C_VEL
LIN {X 0,Y 324.13,Z 576.329,A -85,B 0,C 180,E1 18588.849,E2 18588.849} C_VEL
LIN {X 0,Y 323.767,Z 589.019,A -85,B 0,C 180,E1 18589.169,E2 18589.169} C_VEL
LIN {X 0,Y 317.855,Z 728.71,A -85,B 0,C 180,E1 18592.321,E2 18592.321} C_VEL
LIN {X 0,Y 316.06,Z 746.976,A -85,B 0,C 180,E1 18593.019,E2 18593.019} C_VEL
LIN {X 0,Y 313.559,Z 764.013,A -85,B 0,C 180,E1 18593.962,E2 18593.962} C_VEL
LIN {X 0,Y 310.477,Z 780.996,A -85,B 0,C 180,E1 18595.249,E2 18595.249} C_VEL
LIN {X 0,Y 307.076,Z 797.055,A -85,B 0,C 180,E1 18596.838,E2 18596.838} C_VEL
LIN {X 0,Y 303.367,Z 812.931,A -85,B 0,C 180,E1 18598.839,E2 18598.839} C_VEL
LIN {X 0,Y 299.66,Z 827.631,A -85,B 0,C 180,E1 18601.175,E2 18601.175} C_VEL
LIN {X 0,Y 296.339,Z 840.776,A -85,B 0,C 180,E1 18603.769,E2 18603.769} C_VEL
LIN {X 0,Y 293.383,Z 852.859,A -85,B 0,C 180,E1 18606.714,E2 18606.714} C_VEL
LIN {X 0,Y 291.087,Z 863.431,A -85,B 0,C 180,E1 18609.911,E2 18609.911} C_VEL
LIN {X 0,Y 289.554,Z 872.487,A -85,B 0,C 180,E1 18613.345,E2 18613.345} C_VEL
LIN {X 0,Y 288.848,Z 879.928,A -85,B 0,C 180,E1 18616.997,E2 18616.997} C_VEL
LIN {X 0,Y 288.89,Z 885.378,A -85,B 0,C 180,E1 18620.639,E2 18620.639} C_VEL
LIN {X 0,Y 289.373,Z 888.813,A -85,B 0,C 180,E1 18624.051,E2 18624.051} C_VEL
LIN {X 0,Y 289.89,Z 890.546,A -85,B 0,C 180,E1 18627.233,E2 18627.233} C_VEL
LIN {X 0,Y 290.122,Z 890.761,A -85,B 0,C 180,E1 18630.198,E2 18630.198} C_VEL
LIN {X 0,Y 289.951,Z 889.614,A -85,B 0,C 180,E1 18633.163,E2 18633.163} C_VEL
LIN {X 0,Y 289.488,Z 886.885,A -85,B 0,C 180,E1 18636.346,E2 18636.346} C_VEL
LIN {X 0,Y 289.079,Z 882.236,A -85,B 0,C 180,E1 18639.758,E2 18639.758} C_VEL
LIN {X 0,Y 289.064,Z 875.706,A -85,B 0,C 180,E1 18643.197,E2 18643.197} C_VEL
LIN {X 0,Y 289.613,Z 867.688,A -85,B 0,C 180,E1 18646.445,E2 18646.445} C_VEL
LIN {X 0,Y 290.838,Z 857.615,A -85,B 0,C 180,E1 18649.689,E2 18649.689} C_VEL
LIN {X 0,Y 292.688,Z 845.911,A -85,B 0,C 180,E1 18652.708,E2 18652.708} C_VEL
LIN {X 0,Y 294.959,Z 833.027,A -85,B 0,C 180,E1 18655.393,E2 18655.393} C_VEL
LIN {X 0,Y 297.608,Z 818.55,A -85,B 0,C 180,E1 18657.84,E2 18657.84} C_VEL
LIN {X 0,Y 300.388,Z 803.004,A -85,B 0,C 180,E1 18659.953,E2 18659.953} C_VEL
LIN {X 0,Y 302.984,Z 787.34,A -85,B 0,C 180,E1 18661.649,E2 18661.649} C_VEL
LIN {X 0,Y 305.47,Z 770.429,A -85,B 0,C 180,E1 18663.078,E2 18663.078} C_VEL
LIN {X 0,Y 307.652,Z 752.53,A -85,B 0,C 180,E1 18664.19,E2 18664.19} C_VEL
LIN {X 0,Y 309.2,Z 734.31,A -85,B 0,C 180,E1 18664.972,E2 18664.972} C_VEL
LIN {X 0,Y 310.129,Z 710.6,A -85,B 0,C 180,E1 18665.58,E2 18665.58} C_VEL
LIN {X 0,Y 314.284,Z 574.775,A -85,B 0,C 180,E1 18668.598,E2 18668.598} C_VEL
LIN {X 0,Y 311.627,Z 542.856,A -85,B 0,C 180,E1 18669.74,E2 18669.74} C_VEL
LIN {X 0,Y 313.575,Z 532.152,A -85,B 0,C 180,E1 18671.193,E2 18671.193} C_VEL
LIN {X 0,Y 307.924,Z 513.621,A -85,B 0,C 180,E1 18674.939,E2 18674.939} C_VEL
LIN {X 0,Y 302.371,Z 497.302,A -85,B 0,C 180,E1 18678.645,E2 18678.645} C_VEL
LIN {X 0,Y 297.067,Z 483.327,A -85,B 0,C 180,E1 18682.225,E2 18682.225} C_VEL
LIN {X 0,Y 292.743,Z 472.899,A -85,B 0,C 180,E1 18685.223,E2 18685.223} C_VEL
LIN {X 0,Y 290.372,Z 466.779,A -85,B 0,C 180,E1 18687.16,E2 18687.16} C_VEL
LIN {X 0,Y 290.366,Z 466.608,A -85,B 0,C 180,E1 18691.827,E2 18691.827} C_VEL
LIN {X 0,Y 290.344,Z 466.62,A -85,B 0,C 180,E1 18696.455,E2 18696.455} C_VEL
LIN {X 0,Y 290.343,Z 466.632,A -85,B 0,C 180,E1 18701.268,E2 18701.268} C_VEL
LIN {X 0,Y 290.362,Z 466.595,A -85,B 0,C 180,E1 18705.849,E2 18705.849} C_VEL
LIN {X 0,Y 290.339,Z 466.599,A -85,B 0,C 180,E1 18710.486,E2 18710.486} C_VEL
LIN {X 0,Y 290.327,Z 466.628,A -85,B 0,C 180,E1 18715.061,E2 18715.061} C_VEL
LIN {X 0,Y 290.325,Z 466.582,A -85,B 0,C 180,E1 18719.606,E2 18719.606} C_VEL
LIN {X 0,Y 290.343,Z 466.629,A -85,B 0,C 180,E1 18724.148,E2 18724.148} C_VEL
LIN {X 0,Y 290.331,Z 466.576,A -85,B 0,C 180,E1 18728.737,E2 18728.737} C_VEL
LIN {X 0,Y 290.317,Z 466.633,A -85,B 0,C 180,E1 18733.342,E2 18733.342} C_VEL
LIN {X 0,Y 290.321,Z 466.578,A -85,B 0,C 180,E1 18738.094,E2 18738.094} C_VEL
LIN {X 0,Y 290.351,Z 466.626,A -85,B 0,C 180,E1 18742.687,E2 18742.687} C_VEL
LIN {X 0,Y 290.312,Z 466.589,A -85,B 0,C 180,E1 18747.305,E2 18747.305} C_VEL
LIN {X 0,Y 290.304,Z 466.62,A -85,B 0,C 180,E1 18751.801,E2 18751.801} C_VEL
LIN {X 0,Y 290.307,Z 466.613,A -85,B 0,C 180,E1 18756.328,E2 18756.328} C_VEL
LIN {X 0,Y 290.327,Z 466.596,A -85,B 0,C 180,E1 18760.87,E2 18760.87} C_VEL
LIN {X 0,Y 290.311,Z 466.63,A -85,B 0,C 180,E1 18765.474,E2 18765.474} C_VEL
LIN {X 0,Y 290.292,Z 466.638,A -85,B 0,C 180,E1 18770.183,E2 18770.183} C_VEL
LIN {X 0,Y 290.306,Z 466.627,A -85,B 0,C 180,E1 18774.888,E2 18774.888} C_VEL
LIN {X 0,Y 290.321,Z 466.864,A -85,B 0,C 180,E1 18778.433,E2 18778.433} C_VEL
LIN {X 0,Y 294.249,Z 477.546,A -85,B 0,C 180,E1 18782.066,E2 18782.066} C_VEL
LIN {X 0,Y 298.371,Z 489.422,A -85,B 0,C 180,E1 18785.713,E2 18785.713} C_VEL
LIN {X 0,Y 302.439,Z 502.954,A -85,B 0,C 180,E1 18789.486,E2 18789.486} C_VEL
LIN {X 0,Y 306.278,Z 517.889,A -85,B 0,C 180,E1 18793.304,E2 18793.304} C_VEL
LIN {X 0,Y 307.854,Z 525.59,A -85,B 0,C 180,E1 18795.132,E2 18795.132} C_VEL
LIN {X 0,Y 303.284,Z 552.091,A -85,B 0,C 180,E1 18800.033,E2 18800.033} C_VEL
LIN {X 0,Y 304.247,Z 559.288,A -85,B 0,C 180,E1 18800.404,E2 18800.404} C_VEL
LIN {X 0,Y 309.731,Z 596.312,A -85,B 0,C 180,E1 18801.971,E2 18801.971} C_VEL
LIN {X 0,Y 306.572,Z 686.553,A -85,B 0,C 180,E1 18804.179,E2 18804.179} C_VEL
LIN {X 0,Y 305.585,Z 703.524,A -85,B 0,C 180,E1 18804.961,E2 18804.961} C_VEL
LIN {X 0,Y 304.286,Z 717.981,A -85,B 0,C 180,E1 18805.948,E2 18805.948} C_VEL
LIN {X 0,Y 302.493,Z 733.079,A -85,B 0,C 180,E1 18807.347,E2 18807.347} C_VEL
LIN {X 0,Y 300.562,Z 746.32,A -85,B 0,C 180,E1 18808.951,E2 18808.951} C_VEL
LIN {X 0,Y 298.422,Z 759.289,A -85,B 0,C 180,E1 18810.96,E2 18810.96} C_VEL
LIN {X 0,Y 298.003,Z 761.625,A -85,B 0,C 180,E1 18811.383,E2 18811.383} C_VEL
LIN {X 0,Y 296.07,Z 767.156,A -85,B 0,C 180,E1 18812.378,E2 18812.378} C_VEL
LIN {X 0,Y 289.63,Z 777.318,A -85,B 0,C 180,E1 18814.345,E2 18814.345} C_VEL
LIN {X 0,Y 286.706,Z 782.56,A -85,B 0,C 180,E1 18815.648,E2 18815.648} C_VEL
LIN {X 0,Y 286.153,Z 784.356,A -85,B 0,C 180,E1 18816.19,E2 18816.19} C_VEL
LIN {X 0,Y 284.649,Z 791.906,A -85,B 0,C 180,E1 18818.891,E2 18818.891} C_VEL
LIN {X 0,Y 283.431,Z 798.392,A -85,B 0,C 180,E1 18822.013,E2 18822.013} C_VEL
LIN {X 0,Y 282.722,Z 802.953,A -85,B 0,C 180,E1 18825.171,E2 18825.171} C_VEL
LIN {X 0,Y 282.464,Z 805.854,A -85,B 0,C 180,E1 18828.577,E2 18828.577} C_VEL
LIN {X 0,Y 282.654,Z 806.814,A -85,B 0,C 180,E1 18831.803,E2 18831.803} C_VEL
LIN {X 0,Y 283.368,Z 805.974,A -85,B 0,C 180,E1 18835.274,E2 18835.274} C_VEL
LIN {X 0,Y 284.605,Z 803.297,A -85,B 0,C 180,E1 18838.541,E2 18838.541} C_VEL
LIN {X 0,Y 286.499,Z 798.696,A -85,B 0,C 180,E1 18841.801,E2 18841.801} C_VEL
LIN {X 0,Y 288.883,Z 792.345,A -85,B 0,C 180,E1 18844.825,E2 18844.825} C_VEL
LIN {X 0,Y 291.735,Z 784.313,A -85,B 0,C 180,E1 18847.654,E2 18847.654} C_VEL
LIN {X 0,Y 294.953,Z 774.354,A -85,B 0,C 180,E1 18850.294,E2 18850.294} C_VEL
LIN {X 0,Y 298.175,Z 763.322,A -85,B 0,C 180,E1 18852.57,E2 18852.57} C_VEL
LIN {X 0,Y 301.356,Z 750.959,A -85,B 0,C 180,E1 18854.552,E2 18854.552} C_VEL
LIN {X 0,Y 304.208,Z 738.129,A -85,B 0,C 180,E1 18856.169,E2 18856.169} C_VEL
LIN {X 0,Y 306.794,Z 723.575,A -85,B 0,C 180,E1 18857.574,E2 18857.574} C_VEL
LIN {X 0,Y 308.876,Z 708.279,A -85,B 0,C 180,E1 18858.677,E2 18858.677} C_VEL
LIN {X 0,Y 310.319,Z 691.879,A -85,B 0,C 180,E1 18859.482,E2 18859.482} C_VEL
LIN {X 0,Y 311.632,Z 665.878,A -85,B 0,C 180,E1 18860.226,E2 18860.226} C_VEL
LIN {X 0,Y 314.827,Z 599.857,A -85,B 0,C 180,E1 18861.85,E2 18861.85} C_VEL
LIN {X 0,Y 310.29,Z 572.16,A -85,B 0,C 180,E1 18863.535,E2 18863.535} C_VEL
LIN {X 0,Y 306.409,Z 551.922,A -85,B 0,C 180,E1 18864.989,E2 18864.989} C_VEL
LIN {X 0,Y 308.992,Z 541.166,A -85,B 0,C 180,E1 18867.069,E2 18867.069} C_VEL
LIN {X 0,Y 306.614,Z 529.703,A -85,B 0,C 180,E1 18870.537,E2 18870.537} C_VEL
LIN {X 0,Y 303.76,Z 518.94,A -85,B 0,C 180,E1 18874.247,E2 18874.247} C_VEL
LIN {X 0,Y 300.663,Z 509.343,A -85,B 0,C 180,E1 18878.096,E2 18878.096} C_VEL
LIN {X 0,Y 297.829,Z 501.325,A -85,B 0,C 180,E1 18881.818,E2 18881.818} C_VEL
LIN {X 0,Y 295.153,Z 494.376,A -85,B 0,C 180,E1 18885.682,E2 18885.682} C_VEL
LIN {X 0,Y 293.215,Z 490.068,A -85,B 0,C 180,E1 18888.592,E2 18888.592} C_VEL
LIN {X 0,Y 291.518,Z 486.099,A -85,B 0,C 180,E1 18891.717,E2 18891.717} C_VEL
LIN {X 0,Y 289.675,Z 481.984,A -85,B 0,C 180,E1 18895.843,E2 18895.843} C_VEL
LIN {X 0,Y 287.836,Z 477.919,A -85,B 0,C 180,E1 18902.787,E2 18902.787} C_VEL
LIN {X 0,Y 287.387,Z 477.318,A -85,B 0,C 180,E1 18907.798,E2 18907.798} C_VEL
LIN {X 0,Y 288.004,Z 478.108,A -85,B 0,C 180,E1 18912.43,E2 18912.43} C_VEL
LIN {X 0,Y 290.573,Z 483.02,A -85,B 0,C 180,E1 18919.917,E2 18919.917} C_VEL
LIN {X 0,Y 293.014,Z 488.213,A -85,B 0,C 180,E1 18924.386,E2 18924.386} C_VEL
LIN {X 0,Y 295.166,Z 492.718,A -85,B 0,C 180,E1 18927.439,E2 18927.439} C_VEL
LIN {X 0,Y 297.354,Z 497.63,A -85,B 0,C 180,E1 18930.213,E2 18930.213} C_VEL
LIN {X 0,Y 299.276,Z 501.872,A -85,B 0,C 180,E1 18932.313,E2 18932.313} C_VEL
LIN {X 0,Y 302.316,Z 508.853,A -85,B 0,C 180,E1 18935.365,E2 18935.365} C_VEL
LIN {X 0,Y 306.056,Z 518.246,A -85,B 0,C 180,E1 18938.847,E2 18938.847} C_VEL
LIN {X 0,Y 310.081,Z 529.61,A -85,B 0,C 180,E1 18942.404,E2 18942.404} C_VEL
LIN {X 0,Y 313.66,Z 541.446,A -85,B 0,C 180,E1 18945.565,E2 18945.565} C_VEL
LIN {X 0,Y 314.672,Z 544.722,A -85,B 0,C 180,E1 18946.292,E2 18946.292} C_VEL
LIN {X 0,Y 315.329,Z 546.733,A -85,B 0,C 180,E1 18946.48,E2 18946.48} C_VEL
LIN {X 0,Y 318.142,Z 577.829,A -85,B 0,C 180,E1 18947.941,E2 18947.941} C_VEL
LIN {X 0,Y 311.571,Z 728.066,A -85,B 0,C 180,E1 18951.409,E2 18951.409} C_VEL
LIN {X 0,Y 309.715,Z 746.256,A -85,B 0,C 180,E1 18952.112,E2 18952.112} C_VEL
LIN {X 0,Y 307.084,Z 763.472,A -85,B 0,C 180,E1 18953.078,E2 18953.078} C_VEL
LIN {X 0,Y 303.87,Z 780.389,A -85,B 0,C 180,E1 18954.381,E2 18954.381} C_VEL
LIN {X 0,Y 300.296,Z 796.496,A -85,B 0,C 180,E1 18956.002,E2 18956.002} C_VEL
LIN {X 0,Y 296.636,Z 811.347,A -85,B 0,C 180,E1 18957.903,E2 18957.903} C_VEL
LIN {X 0,Y 292.816,Z 825.759,A -85,B 0,C 180,E1 18960.21,E2 18960.21} C_VEL
LIN {X 0,Y 289.227,Z 838.992,A -85,B 0,C 180,E1 18962.85,E2 18962.85} C_VEL
LIN {X 0,Y 286.03,Z 851.187,A -85,B 0,C 180,E1 18965.859,E2 18965.859} C_VEL
LIN {X 0,Y 283.466,Z 862.003,A -85,B 0,C 180,E1 18969.183,E2 18969.183} C_VEL
LIN {X 0,Y 281.774,Z 870.992,A -85,B 0,C 180,E1 18972.659,E2 18972.659} C_VEL
LIN {X 0,Y 280.911,Z 878.527,A -85,B 0,C 180,E1 18976.414,E2 18976.414} C_VEL
LIN {X 0,Y 280.88,Z 884.035,A -85,B 0,C 180,E1 18980.162,E2 18980.162} C_VEL
LIN {X 0,Y 281.357,Z 887.532,A -85,B 0,C 180,E1 18983.676,E2 18983.676} C_VEL
LIN {X 0,Y 281.926,Z 889.33,A -85,B 0,C 180,E1 18986.951,E2 18986.951} C_VEL
LIN {X 0,Y 282.215,Z 889.591,A -85,B 0,C 180,E1 18990,E2 18990} C_VEL
LIN {X 0,Y 282.046,Z 888.488,A -85,B 0,C 180,E1 18993.049,E2 18993.049} C_VEL
LIN {X 0,Y 281.555,Z 885.793,A -85,B 0,C 180,E1 18996.321,E2 18996.321} C_VEL
LIN {X 0,Y 281.118,Z 881.111,A -85,B 0,C 180,E1 18999.867,E2 18999.867} C_VEL
LIN {X 0,Y 281.103,Z 874.656,A -85,B 0,C 180,E1 19003.368,E2 19003.368} C_VEL
LIN {X 0,Y 281.692,Z 866.637,A -85,B 0,C 180,E1 19006.709,E2 19006.709} C_VEL
LIN {X 0,Y 282.982,Z 856.547,A -85,B 0,C 180,E1 19010.044,E2 19010.044} C_VEL
LIN {X 0,Y 284.927,Z 844.822,A -85,B 0,C 180,E1 19013.143,E2 19013.143} C_VEL
LIN {X 0,Y 287.299,Z 831.92,A -85,B 0,C 180,E1 19015.898,E2 19015.898} C_VEL
LIN {X 0,Y 290.076,Z 817.42,A -85,B 0,C 180,E1 19018.403,E2 19018.403} C_VEL
LIN {X 0,Y 292.97,Z 801.83,A -85,B 0,C 180,E1 19020.565,E2 19020.565} C_VEL
LIN {X 0,Y 295.67,Z 786.099,A -85,B 0,C 180,E1 19022.297,E2 19022.297} C_VEL
LIN {X 0,Y 298.283,Z 768.867,A -85,B 0,C 180,E1 19023.767,E2 19023.767} C_VEL
LIN {X 0,Y 300.496,Z 750.972,A -85,B 0,C 180,E1 19024.883,E2 19024.883} C_VEL
LIN {X 0,Y 302.064,Z 732.635,A -85,B 0,C 180,E1 19025.669,E2 19025.669} C_VEL
LIN {X 0,Y 303.082,Z 706.208,A -85,B 0,C 180,E1 19026.337,E2 19026.337} C_VEL
LIN {X 0,Y 307.263,Z 575.465,A -85,B 0,C 180,E1 19029.304,E2 19029.304} C_VEL
LIN {X 0,Y 304.678,Z 542.693,A -85,B 0,C 180,E1 19030.525,E2 19030.525} C_VEL
LIN {X 0,Y 306.261,Z 534.775,A -85,B 0,C 180,E1 19031.615,E2 19031.615} C_VEL
LIN {X 0,Y 300.892,Z 516.942,A -85,B 0,C 180,E1 19035.326,E2 19035.326} C_VEL
LIN {X 0,Y 295.609,Z 501.202,A -85,B 0,C 180,E1 19038.991,E2 19038.991} C_VEL
LIN {X 0,Y 290.616,Z 487.865,A -85,B 0,C 180,E1 19042.486,E2 19042.486} C_VEL
LIN {X 0,Y 286.34,Z 477.417,A -85,B 0,C 180,E1 19045.551,E2 19045.551} C_VEL
LIN {X 0,Y 283.322,Z 470.416,A -85,B 0,C 180,E1 19047.8,E2 19047.8} C_VEL
LIN {X 0,Y 282.419,Z 467.705,A -85,B 0,C 180,E1 19048.795,E2 19048.795} C_VEL
LIN {X 0,Y 282.414,Z 467.592,A -85,B 0,C 180,E1 19053.507,E2 19053.507} C_VEL
LIN {X 0,Y 282.414,Z 467.586,A -85,B 0,C 180,E1 19058.177,E2 19058.177} C_VEL
LIN {X 0,Y 282.395,Z 467.6,A -85,B 0,C 180,E1 19062.937,E2 19062.937} C_VEL
LIN {X 0,Y 282.403,Z 467.616,A -85,B 0,C 180,E1 19067.528,E2 19067.528} C_VEL
LIN {X 0,Y 282.413,Z 467.572,A -85,B 0,C 180,E1 19072.269,E2 19072.269} C_VEL
LIN {X 0,Y 282.389,Z 467.616,A -85,B 0,C 180,E1 19076.956,E2 19076.956} C_VEL
LIN {X 0,Y 282.384,Z 467.58,A -85,B 0,C 180,E1 19081.624,E2 19081.624} C_VEL
LIN {X 0,Y 282.41,Z 467.592,A -85,B 0,C 180,E1 19086.302,E2 19086.302} C_VEL
LIN {X 0,Y 282.383,Z 467.593,A -85,B 0,C 180,E1 19091.023,E2 19091.023} C_VEL
LIN {X 0,Y 282.373,Z 467.586,A -85,B 0,C 180,E1 19095.612,E2 19095.612} C_VEL
LIN {X 0,Y 282.392,Z 467.602,A -85,B 0,C 180,E1 19100.304,E2 19100.304} C_VEL
LIN {X 0,Y 282.389,Z 467.577,A -85,B 0,C 180,E1 19104.92,E2 19104.92} C_VEL
LIN {X 0,Y 282.372,Z 467.619,A -85,B 0,C 180,E1 19109.485,E2 19109.485} C_VEL
LIN {X 0,Y 282.367,Z 467.577,A -85,B 0,C 180,E1 19114.265,E2 19114.265} C_VEL
LIN {X 0,Y 282.395,Z 467.614,A -85,B 0,C 180,E1 19118.836,E2 19118.836} C_VEL
LIN {X 0,Y 282.371,Z 467.607,A -85,B 0,C 180,E1 19123.456,E2 19123.456} C_VEL
LIN {X 0,Y 282.35,Z 467.594,A -85,B 0,C 180,E1 19128.044,E2 19128.044} C_VEL
LIN {X 0,Y 282.361,Z 467.599,A -85,B 0,C 180,E1 19132.733,E2 19132.733} C_VEL
LIN {X 0,Y 282.406,Z 467.899,A -85,B 0,C 180,E1 19136.928,E2 19136.928} C_VEL
LIN {X 0,Y 286.427,Z 478.555,A -85,B 0,C 180,E1 19140.775,E2 19140.775} C_VEL
LIN {X 0,Y 290.632,Z 490.657,A -85,B 0,C 180,E1 19144.65,E2 19144.65} C_VEL
LIN {X 0,Y 294.656,Z 503.885,A -85,B 0,C 180,E1 19148.501,E2 19148.501} C_VEL
LIN {X 0,Y 298.382,Z 517.972,A -85,B 0,C 180,E1 19152.245,E2 19152.245} C_VEL
LIN {X 0,Y 300.525,Z 527.724,A -85,B 0,C 180,E1 19154.662,E2 19154.662} C_VEL
LIN {X 0,Y 296.132,Z 552.348,A -85,B 0,C 180,E1 19159.278,E2 19159.278} C_VEL
LIN {X 0,Y 302.69,Z 597.282,A -85,B 0,C 180,E1 19161.269,E2 19161.269} C_VEL
LIN {X 0,Y 299.414,Z 687.07,A -85,B 0,C 180,E1 19163.51,E2 19163.51} C_VEL
LIN {X 0,Y 298.361,Z 704.385,A -85,B 0,C 180,E1 19164.326,E2 19164.326} C_VEL
LIN {X 0,Y 296.918,Z 719.577,A -85,B 0,C 180,E1 19165.4,E2 19165.4} C_VEL
LIN {X 0,Y 295.1,Z 734.183,A -85,B 0,C 180,E1 19166.795,E2 19166.795} C_VEL
LIN {X 0,Y 293.068,Z 747.489,A -85,B 0,C 180,E1 19168.454,E2 19168.454} C_VEL
LIN {X 0,Y 290.86,Z 760.317,A -85,B 0,C 180,E1 19170.492,E2 19170.492} C_VEL
LIN {X 0,Y 288.706,Z 771.593,A -85,B 0,C 180,E1 19172.779,E2 19172.779} C_VEL
LIN {X 0,Y 286.676,Z 781.797,A -85,B 0,C 180,E1 19175.403,E2 19175.403} C_VEL
LIN {X 0,Y 286.153,Z 784.356,A -85,B 0,C 180,E1 19176.19,E2 19176.19} C_VEL
LIN {X 0,Y 284.408,Z 788.463,A -85,B 0,C 180,E1 19177.468,E2 19177.468} C_VEL
LIN {X 0,Y 278.817,Z 795.213,A -85,B 0,C 180,E1 19179.832,E2 19179.832} C_VEL
LIN {X 0,Y 276.033,Z 798.708,A -85,B 0,C 180,E1 19181.429,E2 19181.429} C_VEL
LIN {X 0,Y 275.417,Z 800.224,A -85,B 0,C 180,E1 19182.289,E2 19182.289} C_VEL
LIN {X 0,Y 274.731,Z 804.616,A -85,B 0,C 180,E1 19185.623,E2 19185.623} C_VEL
LIN {X 0,Y 274.544,Z 807.176,A -85,B 0,C 180,E1 19188.912,E2 19188.912} C_VEL
LIN {X 0,Y 274.832,Z 807.994,A -85,B 0,C 180,E1 19192.47,E2 19192.47} C_VEL
LIN {X 0,Y 275.651,Z 806.993,A -85,B 0,C 180,E1 19195.898,E2 19195.898} C_VEL
LIN {X 0,Y 277.116,Z 804.002,A -85,B 0,C 180,E1 19199.386,E2 19199.386} C_VEL
LIN {X 0,Y 279.076,Z 799.521,A -85,B 0,C 180,E1 19202.507,E2 19202.507} C_VEL
LIN {X 0,Y 281.675,Z 793.022,A -85,B 0,C 180,E1 19205.621,E2 19205.621} C_VEL
LIN {X 0,Y 284.655,Z 785.067,A -85,B 0,C 180,E1 19208.441,E2 19208.441} C_VEL
LIN {X 0,Y 288.081,Z 775.031,A -85,B 0,C 180,E1 19211.135,E2 19211.135} C_VEL
LIN {X 0,Y 291.325,Z 764.483,A -85,B 0,C 180,E1 19213.347,E2 19213.347} C_VEL
LIN {X 0,Y 294.774,Z 751.778,A -85,B 0,C 180,E1 19215.423,E2 19215.423} C_VEL
LIN {X 0,Y 297.879,Z 738.421,A -85,B 0,C 180,E1 19217.124,E2 19217.124} C_VEL
LIN {X 0,Y 300.62,Z 723.649,A -85,B 0,C 180,E1 19218.557,E2 19218.557} C_VEL
LIN {X 0,Y 302.781,Z 708.242,A -85,B 0,C 180,E1 19219.665,E2 19219.665} C_VEL
LIN {X 0,Y 304.314,Z 691.324,A -85,B 0,C 180,E1 19220.489,E2 19220.489} C_VEL
LIN {X 0,Y 306.373,Z 652.106,A -85,B 0,C 180,E1 19221.559,E2 19221.559} C_VEL
LIN {X 0,Y 308.91,Z 601.221,A -85,B 0,C 180,E1 19222.824,E2 19222.824} C_VEL
LIN {X 0,Y 304.464,Z 573.452,A -85,B 0,C 180,E1 19224.575,E2 19224.575} C_VEL
LIN {X 0,Y 300.442,Z 552.585,A -85,B 0,C 180,E1 19226.121,E2 19226.121} C_VEL
LIN {X 0,Y 300.693,Z 550.096,A -85,B 0,C 180,E1 19226.496,E2 19226.496} C_VEL
LIN {X 0,Y 302.175,Z 544.219,A -85,B 0,C 180,E1 19227.697,E2 19227.697} C_VEL
LIN {X 0,Y 299.965,Z 533.353,A -85,B 0,C 180,E1 19231.097,E2 19231.097} C_VEL
LIN {X 0,Y 297.252,Z 522.999,A -85,B 0,C 180,E1 19234.799,E2 19234.799} C_VEL
LIN {X 0,Y 294.494,Z 514.065,A -85,B 0,C 180,E1 19238.489,E2 19238.489} C_VEL
LIN {X 0,Y 291.949,Z 506.63,A -85,B 0,C 180,E1 19242.047,E2 19242.047} C_VEL
LIN {X 0,Y 289.318,Z 499.722,A -85,B 0,C 180,E1 19246,E2 19246} C_VEL
LIN {X 0,Y 287.605,Z 495.71,A -85,B 0,C 180,E1 19248.773,E2 19248.773} C_VEL
LIN {X 0,Y 285.964,Z 491.796,A -85,B 0,C 180,E1 19251.96,E2 19251.96} C_VEL
LIN {X 0,Y 284.323,Z 487.912,A -85,B 0,C 180,E1 19255.966,E2 19255.966} C_VEL
LIN {X 0,Y 282.651,Z 484.006,A -85,B 0,C 180,E1 19262.838,E2 19262.838} C_VEL
LIN {X 0,Y 282.265,Z 483.463,A -85,B 0,C 180,E1 19267.94,E2 19267.94} C_VEL
LIN {X 0,Y 282.89,Z 484.282,A -85,B 0,C 180,E1 19272.45,E2 19272.45} C_VEL
LIN {X 0,Y 285.359,Z 489.154,A -85,B 0,C 180,E1 19279.869,E2 19279.869} C_VEL
LIN {X 0,Y 287.68,Z 494.128,A -85,B 0,C 180,E1 19284.212,E2 19284.212} C_VEL
LIN {X 0,Y 289.787,Z 498.665,A -85,B 0,C 180,E1 19287.315,E2 19287.315} C_VEL
LIN {X 0,Y 291.852,Z 503.352,A -85,B 0,C 180,E1 19290.012,E2 19290.012} C_VEL
LIN {X 0,Y 294.703,Z 509.556,A -85,B 0,C 180,E1 19293.109,E2 19293.109} C_VEL
LIN {X 0,Y 298.784,Z 519.797,A -85,B 0,C 180,E1 19297.279,E2 19297.279} C_VEL
LIN {X 0,Y 302.573,Z 530.389,A -85,B 0,C 180,E1 19300.866,E2 19300.866} C_VEL
LIN {X 0,Y 306.296,Z 542.355,A -85,B 0,C 180,E1 19304.312,E2 19304.312} C_VEL
LIN {X 0,Y 307.22,Z 545.099,A -85,B 0,C 180,E1 19304.929,E2 19304.929} C_VEL
LIN {X 0,Y 309.792,Z 550.091,A -85,B 0,C 180,E1 19305.585,E2 19305.585} C_VEL
LIN {X 0,Y 312.329,Z 580.199,A -85,B 0,C 180,E1 19307.026,E2 19307.026} C_VEL
LIN {X 0,Y 305.386,Z 727.258,A -85,B 0,C 180,E1 19310.454,E2 19310.454} C_VEL
LIN {X 0,Y 303.464,Z 745.446,A -85,B 0,C 180,E1 19311.163,E2 19311.163} C_VEL
LIN {X 0,Y 300.688,Z 762.93,A -85,B 0,C 180,E1 19312.157,E2 19312.157} C_VEL
LIN {X 0,Y 297.278,Z 780.07,A -85,B 0,C 180,E1 19313.499,E2 19313.499} C_VEL
LIN {X 0,Y 293.631,Z 795.733,A -85,B 0,C 180,E1 19315.106,E2 19315.106} C_VEL
LIN {X 0,Y 289.716,Z 810.825,A -85,B 0,C 180,E1 19317.074,E2 19317.074} C_VEL
LIN {X 0,Y 285.598,Z 825.498,A -85,B 0,C 180,E1 19319.494,E2 19319.494} C_VEL
LIN {X 0,Y 281.947,Z 838.164,A -85,B 0,C 180,E1 19322.089,E2 19322.089} C_VEL
LIN {X 0,Y 278.547,Z 850.277,A -85,B 0,C 180,E1 19325.167,E2 19325.167} C_VEL
LIN {X 0,Y 275.822,Z 860.883,A -85,B 0,C 180,E1 19328.523,E2 19328.523} C_VEL
LIN {X 0,Y 273.942,Z 869.988,A -85,B 0,C 180,E1 19332.146,E2 19332.146} C_VEL
LIN {X 0,Y 272.991,Z 877.116,A -85,B 0,C 180,E1 19335.795,E2 19335.795} C_VEL
LIN {X 0,Y 272.873,Z 882.699,A -85,B 0,C 180,E1 19339.657,E2 19339.657} C_VEL
LIN {X 0,Y 273.332,Z 886.257,A -85,B 0,C 180,E1 19343.278,E2 19343.278} C_VEL
LIN {X 0,Y 273.956,Z 888.105,A -85,B 0,C 180,E1 19346.653,E2 19346.653} C_VEL
LIN {X 0,Y 274.293,Z 888.415,A -85,B 0,C 180,E1 19349.792,E2 19349.792} C_VEL
LIN {X 0,Y 274.142,Z 887.359,A -85,B 0,C 180,E1 19352.927,E2 19352.927} C_VEL
LIN {X 0,Y 273.621,Z 884.671,A -85,B 0,C 180,E1 19356.315,E2 19356.315} C_VEL
LIN {X 0,Y 273.163,Z 880.084,A -85,B 0,C 180,E1 19359.907,E2 19359.907} C_VEL
LIN {X 0,Y 273.146,Z 873.571,A -85,B 0,C 180,E1 19363.549,E2 19363.549} C_VEL
LIN {X 0,Y 273.775,Z 865.558,A -85,B 0,C 180,E1 19366.988,E2 19366.988} C_VEL
LIN {X 0,Y 275.136,Z 855.468,A -85,B 0,C 180,E1 19370.419,E2 19370.419} C_VEL
LIN {X 0,Y 277.184,Z 843.733,A -85,B 0,C 180,E1 19373.604,E2 19373.604} C_VEL
LIN {X 0,Y 279.667,Z 830.813,A -85,B 0,C 180,E1 19376.431,E2 19376.431} C_VEL
LIN {X 0,Y 282.572,Z 816.288,A -85,B 0,C 180,E1 19378.997,E2 19378.997} C_VEL
LIN {X 0,Y 285.441,Z 801.426,A -85,B 0,C 180,E1 19381.11,E2 19381.11} C_VEL
LIN {X 0,Y 288.351,Z 785.118,A -85,B 0,C 180,E1 19382.951,E2 19382.951} C_VEL
LIN {X 0,Y 291,Z 768.275,A -85,B 0,C 180,E1 19384.418,E2 19384.418} C_VEL
LIN {X 0,Y 293.282,Z 750.41,A -85,B 0,C 180,E1 19385.555,E2 19385.555} C_VEL
LIN {X 0,Y 294.897,Z 732.077,A -85,B 0,C 180,E1 19386.357,E2 19386.357} C_VEL
LIN {X 0,Y 295.953,Z 705.758,A -85,B 0,C 180,E1 19387.036,E2 19387.036} C_VEL
LIN {X 0,Y 300.279,Z 576.321,A -85,B 0,C 180,E1 19390.027,E2 19390.027} C_VEL
LIN {X 0,Y 297.697,Z 543.033,A -85,B 0,C 180,E1 19391.286,E2 19391.286} C_VEL
LIN {X 0,Y 298.803,Z 536.851,A -85,B 0,C 180,E1 19392.168,E2 19392.168} C_VEL
LIN {X 0,Y 293.513,Z 519.168,A -85,B 0,C 180,E1 19395.979,E2 19395.979} C_VEL
LIN {X 0,Y 288.206,Z 503.251,A -85,B 0,C 180,E1 19399.814,E2 19399.814} C_VEL
LIN {X 0,Y 283.032,Z 489.483,A -85,B 0,C 180,E1 19403.595,E2 19403.595} C_VEL
LIN {X 0,Y 278.864,Z 479.31,A -85,B 0,C 180,E1 19406.731,E2 19406.731} C_VEL
LIN {X 0,Y 275.636,Z 471.85,A -85,B 0,C 180,E1 19409.285,E2 19409.285} C_VEL
LIN {X 0,Y 274.483,Z 468.723,A -85,B 0,C 180,E1 19410.49,E2 19410.49} C_VEL
LIN {X 0,Y 274.469,Z 468.606,A -85,B 0,C 180,E1 19415.233,E2 19415.233} C_VEL
LIN {X 0,Y 274.477,Z 468.585,A -85,B 0,C 180,E1 19419.976,E2 19419.976} C_VEL
LIN {X 0,Y 274.453,Z 468.569,A -85,B 0,C 180,E1 19424.794,E2 19424.794} C_VEL
LIN {X 0,Y 274.46,Z 468.592,A -85,B 0,C 180,E1 19429.615,E2 19429.615} C_VEL
LIN {X 0,Y 274.469,Z 468.588,A -85,B 0,C 180,E1 19434.356,E2 19434.356} C_VEL
LIN {X 0,Y 274.442,Z 468.561,A -85,B 0,C 180,E1 19439.165,E2 19439.165} C_VEL
LIN {X 0,Y 274.459,Z 468.606,A -85,B 0,C 180,E1 19443.969,E2 19443.969} C_VEL
LIN {X 0,Y 274.459,Z 468.55,A -85,B 0,C 180,E1 19448.59,E2 19448.59} C_VEL
LIN {X 0,Y 274.44,Z 468.611,A -85,B 0,C 180,E1 19453.484,E2 19453.484} C_VEL
LIN {X 0,Y 274.449,Z 468.553,A -85,B 0,C 180,E1 19458.259,E2 19458.259} C_VEL
LIN {X 0,Y 274.455,Z 468.603,A -85,B 0,C 180,E1 19462.943,E2 19462.943} C_VEL
LIN {X 0,Y 274.429,Z 468.572,A -85,B 0,C 180,E1 19467.799,E2 19467.799} C_VEL
LIN {X 0,Y 274.437,Z 468.581,A -85,B 0,C 180,E1 19472.383,E2 19472.383} C_VEL
LIN {X 0,Y 274.446,Z 468.604,A -85,B 0,C 180,E1 19477.073,E2 19477.073} C_VEL
LIN {X 0,Y 274.421,Z 468.574,A -85,B 0,C 180,E1 19481.675,E2 19481.675} C_VEL
LIN {X 0,Y 274.422,Z 468.588,A -85,B 0,C 180,E1 19486.478,E2 19486.478} C_VEL
LIN {X 0,Y 274.45,Z 468.601,A -85,B 0,C 180,E1 19491.228,E2 19491.228} C_VEL
LIN {X 0,Y 274.473,Z 468.878,A -85,B 0,C 180,E1 19495.27,E2 19495.27} C_VEL
LIN {X 0,Y 278.644,Z 479.834,A -85,B 0,C 180,E1 19499.452,E2 19499.452} C_VEL
LIN {X 0,Y 282.83,Z 491.619,A -85,B 0,C 180,E1 19503.433,E2 19503.433} C_VEL
LIN {X 0,Y 286.689,Z 504.011,A -85,B 0,C 180,E1 19507.224,E2 19507.224} C_VEL
LIN {X 0,Y 290.481,Z 518.317,A -85,B 0,C 180,E1 19511.188,E2 19511.188} C_VEL
LIN {X 0,Y 293.125,Z 530.378,A -85,B 0,C 180,E1 19514.265,E2 19514.265} C_VEL
LIN {X 0,Y 289.033,Z 552.435,A -85,B 0,C 180,E1 19518.465,E2 19518.465} C_VEL
LIN {X 0,Y 295.654,Z 598.37,A -85,B 0,C 180,E1 19520.55,E2 19520.55} C_VEL
LIN {X 0,Y 292.259,Z 687.74,A -85,B 0,C 180,E1 19522.826,E2 19522.826} C_VEL
LIN {X 0,Y 291.155,Z 705.166,A -85,B 0,C 180,E1 19523.666,E2 19523.666} C_VEL
LIN {X 0,Y 289.666,Z 720.21,A -85,B 0,C 180,E1 19524.751,E2 19524.751} C_VEL
LIN {X 0,Y 287.727,Z 735.191,A -85,B 0,C 180,E1 19526.214,E2 19526.214} C_VEL
LIN {X 0,Y 285.516,Z 749.021,A -85,B 0,C 180,E1 19527.993,E2 19527.993} C_VEL
LIN {X 0,Y 283.208,Z 761.846,A -85,B 0,C 180,E1 19530.101,E2 19530.101} C_VEL
LIN {X 0,Y 280.976,Z 773.008,A -85,B 0,C 180,E1 19532.447,E2 19532.447} C_VEL
LIN {X 0,Y 278.873,Z 783.132,A -85,B 0,C 180,E1 19535.142,E2 19535.142} C_VEL
LIN {X 0,Y 277.089,Z 791.609,A -85,B 0,C 180,E1 19538.09,E2 19538.09} C_VEL
LIN {X 0,Y 275.801,Z 798.12,A -85,B 0,C 180,E1 19541.077,E2 19541.077} C_VEL
LIN {X 0,Y 275.417,Z 800.224,A -85,B 0,C 180,E1 19542.289,E2 19542.289} C_VEL
LIN {X 0,Y 274.056,Z 802.648,A -85,B 0,C 180,E1 19543.802,E2 19543.802} C_VEL
LIN {X 0,Y 269.231,Z 806.416,A -85,B 0,C 180,E1 19546.59,E2 19546.59} C_VEL
LIN {X 0,Y 266.89,Z 808.069,A -85,B 0,C 180,E1 19548.526,E2 19548.526} C_VEL
LIN {X 0,Y 266.629,Z 808.493,A -85,B 0,C 180,E1 19549.356,E2 19549.356} C_VEL
LIN {X 0,Y 266.994,Z 809.179,A -85,B 0,C 180,E1 19552.921,E2 19552.921} C_VEL
LIN {X 0,Y 267.904,Z 808.078,A -85,B 0,C 180,E1 19556.398,E2 19556.398} C_VEL
LIN {X 0,Y 269.562,Z 804.954,A -85,B 0,C 180,E1 19560.049,E2 19560.049} C_VEL
LIN {X 0,Y 271.695,Z 800.333,A -85,B 0,C 180,E1 19563.252,E2 19563.252} C_VEL
LIN {X 0,Y 274.492,Z 793.781,A -85,B 0,C 180,E1 19566.422,E2 19566.422} C_VEL
LIN {X 0,Y 277.702,Z 785.656,A -85,B 0,C 180,E1 19569.322,E2 19569.322} C_VEL
LIN {X 0,Y 281.292,Z 775.736,A -85,B 0,C 180,E1 19572.02,E2 19572.02} C_VEL
LIN {X 0,Y 284.797,Z 764.867,A -85,B 0,C 180,E1 19574.318,E2 19574.318} C_VEL
LIN {X 0,Y 288.447,Z 752.054,A -85,B 0,C 180,E1 19576.424,E2 19576.424} C_VEL
LIN {X 0,Y 291.58,Z 739.095,A -85,B 0,C 180,E1 19578.083,E2 19578.083} C_VEL
LIN {X 0,Y 294.548,Z 723.751,A -85,B 0,C 180,E1 19579.581,E2 19579.581} C_VEL
LIN {X 0,Y 296.757,Z 708.441,A -85,B 0,C 180,E1 19580.68,E2 19580.68} C_VEL
LIN {X 0,Y 298.344,Z 691.575,A -85,B 0,C 180,E1 19581.503,E2 19581.503} C_VEL
LIN {X 0,Y 300.994,Z 643.287,A -85,B 0,C 180,E1 19582.809,E2 19582.809} C_VEL
LIN {X 0,Y 303.085,Z 602.585,A -85,B 0,C 180,E1 19583.835,E2 19583.835} C_VEL
LIN {X 0,Y 298.799,Z 575.104,A -85,B 0,C 180,E1 19585.634,E2 19585.634} C_VEL
LIN {X 0,Y 294.535,Z 551.846,A -85,B 0,C 180,E1 19587.448,E2 19587.448} C_VEL
LIN {X 0,Y 295.447,Z 547.686,A -85,B 0,C 180,E1 19588.236,E2 19588.236} C_VEL
LIN {X 0,Y 293.323,Z 536.917,A -85,B 0,C 180,E1 19591.717,E2 19591.717} C_VEL
LIN {X 0,Y 290.783,Z 526.989,A -85,B 0,C 180,E1 19595.413,E2 19595.413} C_VEL
LIN {X 0,Y 288.126,Z 517.996,A -85,B 0,C 180,E1 19599.27,E2 19599.27} C_VEL
LIN {X 0,Y 285.626,Z 510.871,A -85,B 0,C 180,E1 19602.899,E2 19602.899} C_VEL
LIN {X 0,Y 283.51,Z 505.074,A -85,B 0,C 180,E1 19606.332,E2 19606.332} C_VEL
LIN {X 0,Y 281.896,Z 501.147,A -85,B 0,C 180,E1 19609.164,E2 19609.164} C_VEL
LIN {X 0,Y 280.544,Z 497.676,A -85,B 0,C 180,E1 19612.01,E2 19612.01} C_VEL
LIN {X 0,Y 278.973,Z 493.842,A -85,B 0,C 180,E1 19616.095,E2 19616.095} C_VEL
LIN {X 0,Y 277.454,Z 490.083,A -85,B 0,C 180,E1 19622.891,E2 19622.891} C_VEL
LIN {X 0,Y 277.124,Z 489.593,A -85,B 0,C 180,E1 19627.88,E2 19627.88} C_VEL
LIN {X 0,Y 277.77,Z 490.456,A -85,B 0,C 180,E1 19632.472,E2 19632.472} C_VEL
LIN {X 0,Y 280.147,Z 495.285,A -85,B 0,C 180,E1 19639.819,E2 19639.819} C_VEL
LIN {X 0,Y 282.349,Z 500.041,A -85,B 0,C 180,E1 19644.031,E2 19644.031} C_VEL
LIN {X 0,Y 284.423,Z 504.637,A -85,B 0,C 180,E1 19647.204,E2 19647.204} C_VEL
LIN {X 0,Y 286.306,Z 508.94,A -85,B 0,C 180,E1 19649.729,E2 19649.729} C_VEL
LIN {X 0,Y 289.068,Z 515.154,A -85,B 0,C 180,E1 19652.891,E2 19652.891} C_VEL
LIN {X 0,Y 292.892,Z 524.991,A -85,B 0,C 180,E1 19656.983,E2 19656.983} C_VEL
LIN {X 0,Y 296.599,Z 535.666,A -85,B 0,C 180,E1 19660.669,E2 19660.669} C_VEL
LIN {X 0,Y 299.3,Z 544.403,A -85,B 0,C 180,E1 19663.259,E2 19663.259} C_VEL
LIN {X 0,Y 304.38,Z 553.943,A -85,B 0,C 180,E1 19664.684,E2 19664.684} C_VEL
LIN {X 0,Y 306.511,Z 581.631,A -85,B 0,C 180,E1 19666.028,E2 19666.028} C_VEL
LIN {X 0,Y 299.331,Z 726.57,A -85,B 0,C 180,E1 19669.451,E2 19669.451} C_VEL
LIN {X 0,Y 297.329,Z 744.744,A -85,B 0,C 180,E1 19670.17,E2 19670.17} C_VEL
LIN {X 0,Y 294.38,Z 762.522,A -85,B 0,C 180,E1 19671.197,E2 19671.197} C_VEL
LIN {X 0,Y 290.885,Z 779.232,A -85,B 0,C 180,E1 19672.526,E2 19672.526} C_VEL
LIN {X 0,Y 287.018,Z 795.072,A -85,B 0,C 180,E1 19674.18,E2 19674.18} C_VEL
LIN {X 0,Y 283.034,Z 809.684,A -85,B 0,C 180,E1 19676.116,E2 19676.116} C_VEL
LIN {X 0,Y 278.752,Z 824.195,A -85,B 0,C 180,E1 19678.541,E2 19678.541} C_VEL
LIN {X 0,Y 274.705,Z 837.402,A -85,B 0,C 180,E1 19681.304,E2 19681.304} C_VEL
LIN {X 0,Y 271.111,Z 849.406,A -85,B 0,C 180,E1 19684.438,E2 19684.438} C_VEL
LIN {X 0,Y 268.183,Z 859.956,A -85,B 0,C 180,E1 19687.88,E2 19687.88} C_VEL
LIN {X 0,Y 266.13,Z 868.992,A -85,B 0,C 180,E1 19691.604,E2 19691.604} C_VEL
LIN {X 0,Y 265.029,Z 876.407,A -85,B 0,C 180,E1 19695.582,E2 19695.582} C_VEL
LIN {X 0,Y 264.897,Z 881.845,A -85,B 0,C 180,E1 19699.562,E2 19699.562} C_VEL
LIN {X 0,Y 265.425,Z 885.414,A -85,B 0,C 180,E1 19703.512,E2 19703.512} C_VEL
LIN {X 0,Y 266.085,Z 887.037,A -85,B 0,C 180,E1 19706.985,E2 19706.985} C_VEL
LIN {X 0,Y 266.388,Z 887.184,A -85,B 0,C 180,E1 19710.215,E2 19710.215} C_VEL
LIN {X 0,Y 266.157,Z 885.865,A -85,B 0,C 180,E1 19713.446,E2 19713.446} C_VEL
LIN {X 0,Y 265.585,Z 882.909,A -85,B 0,C 180,E1 19716.92,E2 19716.92} C_VEL
LIN {X 0,Y 265.159,Z 877.997,A -85,B 0,C 180,E1 19720.648,E2 19720.648} C_VEL
LIN {X 0,Y 265.258,Z 871.169,A -85,B 0,C 180,E1 19724.406,E2 19724.406} C_VEL
LIN {X 0,Y 266.068,Z 862.785,A -85,B 0,C 180,E1 19727.948,E2 19727.948} C_VEL
LIN {X 0,Y 267.545,Z 852.948,A -85,B 0,C 180,E1 19731.255,E2 19731.255} C_VEL
LIN {X 0,Y 269.634,Z 841.75,A -85,B 0,C 180,E1 19734.306,E2 19734.306} C_VEL
LIN {X 0,Y 272.229,Z 828.895,A -85,B 0,C 180,E1 19737.155,E2 19737.155} C_VEL
LIN {X 0,Y 275.283,Z 814.258,A -85,B 0,C 180,E1 19739.765,E2 19739.765} C_VEL
LIN {X 0,Y 278.245,Z 799.408,A -85,B 0,C 180,E1 19741.887,E2 19741.887} C_VEL
LIN {X 0,Y 281.165,Z 783.483,A -85,B 0,C 180,E1 19743.694,E2 19743.694} C_VEL
LIN {X 0,Y 283.893,Z 766.495,A -85,B 0,C 180,E1 19745.171,E2 19745.171} C_VEL
LIN {X 0,Y 286.205,Z 748.642,A -85,B 0,C 180,E1 19746.31,E2 19746.31} C_VEL
LIN {X 0,Y 287.857,Z 729.726,A -85,B 0,C 180,E1 19747.13,E2 19747.13} C_VEL
LIN {X 0,Y 289.171,Z 695.142,A -85,B 0,C 180,E1 19747.994,E2 19747.994} C_VEL
LIN {X 0,Y 293.322,Z 577.057,A -85,B 0,C 180,E1 19750.785,E2 19750.785} C_VEL
LIN {X 0,Y 290.793,Z 543.136,A -85,B 0,C 180,E1 19752.105,E2 19752.105} C_VEL
LIN {X 0,Y 291.527,Z 539.523,A -85,B 0,C 180,E1 19752.621,E2 19752.621} C_VEL
LIN {X 0,Y 286.307,Z 521.895,A -85,B 0,C 180,E1 19756.53,E2 19756.53} C_VEL
LIN {X 0,Y 281.403,Z 506.983,A -85,B 0,C 180,E1 19760.241,E2 19760.241} C_VEL
LIN {X 0,Y 276.297,Z 493.293,A -85,B 0,C 180,E1 19764.11,E2 19764.11} C_VEL
LIN {X 0,Y 271.499,Z 481.224,A -85,B 0,C 180,E1 19767.974,E2 19767.974} C_VEL
LIN {X 0,Y 267.819,Z 473.054,A -85,B 0,C 180,E1 19770.966,E2 19770.966} C_VEL
LIN {X 0,Y 266.545,Z 469.708,A -85,B 0,C 180,E1 19772.37,E2 19772.37} C_VEL
LIN {X 0,Y 266.531,Z 469.568,A -85,B 0,C 180,E1 19777.346,E2 19777.346} C_VEL
LIN {X 0,Y 266.536,Z 469.592,A -85,B 0,C 180,E1 19782.085,E2 19782.085} C_VEL
LIN {X 0,Y 266.516,Z 469.581,A -85,B 0,C 180,E1 19786.992,E2 19786.992} C_VEL
LIN {X 0,Y 266.527,Z 469.549,A -85,B 0,C 180,E1 19791.805,E2 19791.805} C_VEL
LIN {X 0,Y 266.522,Z 469.595,A -85,B 0,C 180,E1 19796.559,E2 19796.559} C_VEL
LIN {X 0,Y 266.504,Z 469.553,A -85,B 0,C 180,E1 19801.505,E2 19801.505} C_VEL
LIN {X 0,Y 266.529,Z 469.567,A -85,B 0,C 180,E1 19806.246,E2 19806.246} C_VEL
LIN {X 0,Y 266.504,Z 469.567,A -85,B 0,C 180,E1 19811.031,E2 19811.031} C_VEL
LIN {X 0,Y 266.5,Z 469.554,A -85,B 0,C 180,E1 19815.896,E2 19815.896} C_VEL
LIN {X 0,Y 266.524,Z 469.584,A -85,B 0,C 180,E1 19820.649,E2 19820.649} C_VEL
LIN {X 0,Y 266.495,Z 469.549,A -85,B 0,C 180,E1 19825.323,E2 19825.323} C_VEL
LIN {X 0,Y 266.498,Z 469.602,A -85,B 0,C 180,E1 19830.182,E2 19830.182} C_VEL
LIN {X 0,Y 266.503,Z 469.554,A -85,B 0,C 180,E1 19835.032,E2 19835.032} C_VEL
LIN {X 0,Y 266.485,Z 469.575,A -85,B 0,C 180,E1 19839.72,E2 19839.72} C_VEL
LIN {X 0,Y 266.492,Z 469.603,A -85,B 0,C 180,E1 19844.557,E2 19844.557} C_VEL
LIN {X 0,Y 266.504,Z 469.579,A -85,B 0,C 180,E1 19849.276,E2 19849.276} C_VEL
LIN {X 0,Y 266.519,Z 469.776,A -85,B 0,C 180,E1 19853.402,E2 19853.402} C_VEL
LIN {X 0,Y 270.802,Z 480.717,A -85,B 0,C 180,E1 19857.881,E2 19857.881} C_VEL
LIN {X 0,Y 274.65,Z 491.511,A -85,B 0,C 180,E1 19861.764,E2 19861.764} C_VEL
LIN {X 0,Y 278.484,Z 503.386,A -85,B 0,C 180,E1 19865.613,E2 19865.613} C_VEL
LIN {X 0,Y 282.373,Z 517.599,A -85,B 0,C 180,E1 19869.777,E2 19869.777} C_VEL
LIN {X 0,Y 285.67,Z 531.704,A -85,B 0,C 180,E1 19873.541,E2 19873.541} C_VEL
LIN {X 0,Y 285.524,Z 534.016,A -85,B 0,C 180,E1 19874.044,E2 19874.044} C_VEL
LIN {X 0,Y 281.99,Z 552.299,A -85,B 0,C 180,E1 19877.585,E2 19877.585} C_VEL
LIN {X 0,Y 288.673,Z 599.354,A -85,B 0,C 180,E1 19879.794,E2 19879.794} C_VEL
LIN {X 0,Y 285.151,Z 688.277,A -85,B 0,C 180,E1 19882.104,E2 19882.104} C_VEL
LIN {X 0,Y 284.002,Z 705.695,A -85,B 0,C 180,E1 19882.96,E2 19882.96} C_VEL
LIN {X 0,Y 282.4,Z 721.225,A -85,B 0,C 180,E1 19884.106,E2 19884.106} C_VEL
LIN {X 0,Y 280.381,Z 736.165,A -85,B 0,C 180,E1 19885.602,E2 19885.602} C_VEL
LIN {X 0,Y 278.079,Z 749.969,A -85,B 0,C 180,E1 19887.424,E2 19887.424} C_VEL
LIN {X 0,Y 275.674,Z 762.791,A -85,B 0,C 180,E1 19889.584,E2 19889.584} C_VEL
LIN {X 0,Y 273.253,Z 774.399,A -85,B 0,C 180,E1 19892.097,E2 19892.097} C_VEL
LIN {X 0,Y 271.225,Z 783.762,A -85,B 0,C 180,E1 19894.652,E2 19894.652} C_VEL
LIN {X 0,Y 269.34,Z 792.34,A -85,B 0,C 180,E1 19897.68,E2 19897.68} C_VEL
LIN {X 0,Y 267.974,Z 798.953,A -85,B 0,C 180,E1 19900.752,E2 19900.752} C_VEL
LIN {X 0,Y 267.045,Z 804.105,A -85,B 0,C 180,E1 19904.129,E2 19904.129} C_VEL
LIN {X 0,Y 266.652,Z 807.393,A -85,B 0,C 180,E1 19907.456,E2 19907.456} C_VEL
LIN {X 0,Y 266.629,Z 808.493,A -85,B 0,C 180,E1 19909.356,E2 19909.356} C_VEL
LIN {X 0,Y 265.752,Z 809.173,A -85,B 0,C 180,E1 19911.012,E2 19911.012} C_VEL
LIN {X 0,Y 261.71,Z 809.896,A -85,B 0,C 180,E1 19914.174,E2 19914.174} C_VEL
LIN {X 0,Y 260.14,Z 809.523,A -85,B 0,C 180,E1 19916.227,E2 19916.227} C_VEL
LIN {X 0,Y 260.189,Z 809.145,A -85,B 0,C 180,E1 19916.958,E2 19916.958} C_VEL
LIN {X 0,Y 261.902,Z 806.158,A -85,B 0,C 180,E1 19920.514,E2 19920.514} C_VEL
LIN {X 0,Y 264.182,Z 801.575,A -85,B 0,C 180,E1 19923.804,E2 19923.804} C_VEL
LIN {X 0,Y 267.278,Z 794.797,A -85,B 0,C 180,E1 19927.172,E2 19927.172} C_VEL
LIN {X 0,Y 270.674,Z 786.683,A -85,B 0,C 180,E1 19930.123,E2 19930.123} C_VEL
LIN {X 0,Y 274.582,Z 776.455,A -85,B 0,C 180,E1 19932.952,E2 19932.952} C_VEL
LIN {X 0,Y 278.36,Z 765.256,A -85,B 0,C 180,E1 19935.333,E2 19935.333} C_VEL
LIN {X 0,Y 282.215,Z 752.33,A -85,B 0,C 180,E1 19937.469,E2 19937.469} C_VEL
LIN {X 0,Y 285.501,Z 739.151,A -85,B 0,C 180,E1 19939.152,E2 19939.152} C_VEL
LIN {X 0,Y 288.577,Z 723.844,A -85,B 0,C 180,E1 19940.649,E2 19940.649} C_VEL
LIN {X 0,Y 290.88,Z 708.222,A -85,B 0,C 180,E1 19941.761,E2 19941.761} C_VEL
LIN {X 0,Y 292.499,Z 691.497,A -85,B 0,C 180,E1 19942.572,E2 19942.572} C_VEL
LIN {X 0,Y 296.161,Z 627.378,A -85,B 0,C 180,E1 19944.279,E2 19944.279} C_VEL
LIN {X 0,Y 297.36,Z 603.967,A -85,B 0,C 180,E1 19944.887,E2 19944.887} C_VEL
LIN {X 0,Y 293.237,Z 576.459,A -85,B 0,C 180,E1 19946.762,E2 19946.762} C_VEL
LIN {X 0,Y 288.814,Z 551.654,A -85,B 0,C 180,E1 19948.77,E2 19948.77} C_VEL
LIN {X 0,Y 288,Z 546.783,A -85,B 0,C 180,E1 19950.219,E2 19950.219} C_VEL
LIN {X 0,Y 285.804,Z 536.551,A -85,B 0,C 180,E1 19953.845,E2 19953.845} C_VEL
LIN {X 0,Y 283.36,Z 527.353,A -85,B 0,C 180,E1 19957.598,E2 19957.598} C_VEL
LIN {X 0,Y 280.95,Z 519.578,A -85,B 0,C 180,E1 19961.319,E2 19961.319} C_VEL
LIN {X 0,Y 278.673,Z 513.031,A -85,B 0,C 180,E1 19965.028,E2 19965.028} C_VEL
LIN {X 0,Y 276.734,Z 507.508,A -85,B 0,C 180,E1 19968.749,E2 19968.749} C_VEL
LIN {X 0,Y 275.025,Z 503.397,A -85,B 0,C 180,E1 19972.269,E2 19972.269} C_VEL
LIN {X 0,Y 273.625,Z 499.772,A -85,B 0,C 180,E1 19976.228,E2 19976.228} C_VEL
LIN {X 0,Y 272.231,Z 496.099,A -85,B 0,C 180,E1 19983.158,E2 19983.158} C_VEL
LIN {X 0,Y 272.017,Z 495.759,A -85,B 0,C 180,E1 19988.454,E2 19988.454} C_VEL
LIN {X 0,Y 272.674,Z 496.735,A -85,B 0,C 180,E1 19992.709,E2 19992.709} C_VEL
LIN {X 0,Y 274.935,Z 501.417,A -85,B 0,C 180,E1 19999.768,E2 19999.768} C_VEL
LIN {X 0,Y 277.022,Z 505.954,A -85,B 0,C 180,E1 20003.843,E2 20003.843} C_VEL
LIN {X 0,Y 279.052,Z 510.571,A -85,B 0,C 180,E1 20007.068,E2 20007.068} C_VEL
LIN {X 0,Y 280.991,Z 515.1,A -85,B 0,C 180,E1 20009.747,E2 20009.747} C_VEL
LIN {X 0,Y 283.598,Z 521.254,A -85,B 0,C 180,E1 20012.884,E2 20012.884} C_VEL
LIN {X 0,Y 287.117,Z 530.52,A -85,B 0,C 180,E1 20016.796,E2 20016.796} C_VEL
LIN {X 0,Y 290.487,Z 540.513,A -85,B 0,C 180,E1 20020.323,E2 20020.323} C_VEL
LIN {X 0,Y 292.07,Z 545.297,A -85,B 0,C 180,E1 20021.746,E2 20021.746} C_VEL
LIN {X 0,Y 299.047,Z 557.773,A -85,B 0,C 180,E1 20023.747,E2 20023.747} C_VEL
LIN {X 0,Y 300.797,Z 582.876,A -85,B 0,C 180,E1 20024.985,E2 20024.985} C_VEL
LIN {X 0,Y 293.357,Z 726.051,A -85,B 0,C 180,E1 20028.412,E2 20028.412} C_VEL
LIN {X 0,Y 291.281,Z 744.152,A -85,B 0,C 180,E1 20029.138,E2 20029.138} C_VEL
LIN {X 0,Y 288.163,Z 762.201,A -85,B 0,C 180,E1 20030.196,E2 20030.196} C_VEL
LIN {X 0,Y 284.525,Z 778.8,A -85,B 0,C 180,E1 20031.538,E2 20031.538} C_VEL
LIN {X 0,Y 280.492,Z 794.549,A -85,B 0,C 180,E1 20033.212,E2 20033.212} C_VEL
LIN {X 0,Y 276.079,Z 809.795,A -85,B 0,C 180,E1 20035.296,E2 20035.296} C_VEL
LIN {X 0,Y 271.647,Z 823.944,A -85,B 0,C 180,E1 20037.744,E2 20037.744} C_VEL
LIN {X 0,Y 267.277,Z 837.383,A -85,B 0,C 180,E1 20040.656,E2 20040.656} C_VEL
LIN {X 0,Y 263.497,Z 849.266,A -85,B 0,C 180,E1 20043.886,E2 20043.886} C_VEL
LIN {X 0,Y 260.416,Z 859.645,A -85,B 0,C 180,E1 20047.422,E2 20047.422} C_VEL
LIN {X 0,Y 258.244,Z 868.472,A -85,B 0,C 180,E1 20051.255,E2 20051.255} C_VEL
LIN {X 0,Y 257.068,Z 875.701,A -85,B 0,C 180,E1 20055.356,E2 20055.356} C_VEL
LIN {X 0,Y 256.921,Z 880.99,A -85,B 0,C 180,E1 20059.461,E2 20059.461} C_VEL
LIN {X 0,Y 257.479,Z 884.426,A -85,B 0,C 180,E1 20063.534,E2 20063.534} C_VEL
LIN {X 0,Y 258.183,Z 885.911,A -85,B 0,C 180,E1 20067.115,E2 20067.115} C_VEL
LIN {X 0,Y 258.48,Z 885.906,A -85,B 0,C 180,E1 20070.444,E2 20070.444} C_VEL
LIN {X 0,Y 258.187,Z 884.482,A -85,B 0,C 180,E1 20073.775,E2 20073.775} C_VEL
LIN {X 0,Y 257.57,Z 881.344,A -85,B 0,C 180,E1 20077.36,E2 20077.36} C_VEL
LIN {X 0,Y 257.174,Z 876.228,A -85,B 0,C 180,E1 20081.21,E2 20081.21} C_VEL
LIN {X 0,Y 257.373,Z 869.123,A -85,B 0,C 180,E1 20085.087,E2 20085.087} C_VEL
LIN {X 0,Y 258.341,Z 860.477,A -85,B 0,C 180,E1 20088.738,E2 20088.738} C_VEL
LIN {X 0,Y 260.148,Z 849.606,A -85,B 0,C 180,E1 20092.365,E2 20092.365} C_VEL
LIN {X 0,Y 262.498,Z 837.919,A -85,B 0,C 180,E1 20095.495,E2 20095.495} C_VEL
LIN {X 0,Y 265.305,Z 824.758,A -85,B 0,C 180,E1 20098.351,E2 20098.351} C_VEL
LIN {X 0,Y 268.375,Z 810.611,A -85,B 0,C 180,E1 20100.816,E2 20100.816} C_VEL
LIN {X 0,Y 271.42,Z 795.617,A -85,B 0,C 180,E1 20102.913,E2 20102.913} C_VEL
LIN {X 0,Y 274.344,Z 779.93,A -85,B 0,C 180,E1 20104.65,E2 20104.65} C_VEL
LIN {X 0,Y 277.18,Z 762.275,A -85,B 0,C 180,E1 20106.142,E2 20106.142} C_VEL
LIN {X 0,Y 279.473,Z 744.377,A -85,B 0,C 180,E1 20107.234,E2 20107.234} C_VEL
LIN {X 0,Y 280.96,Z 725.901,A -85,B 0,C 180,E1 20107.992,E2 20107.992} C_VEL
LIN {X 0,Y 286.417,Z 577.761,A -85,B 0,C 180,E1 20111.581,E2 20111.581} C_VEL
LIN {X 0,Y 283.938,Z 543.332,A -85,B 0,C 180,E1 20112.953,E2 20112.953} C_VEL
LIN {X 0,Y 284.069,Z 541.535,A -85,B 0,C 180,E1 20113.232,E2 20113.232} C_VEL
LIN {X 0,Y 279.12,Z 524.631,A -85,B 0,C 180,E1 20117.109,E2 20117.109} C_VEL
LIN {X 0,Y 274.249,Z 509.753,A -85,B 0,C 180,E1 20120.947,E2 20120.947} C_VEL
LIN {X 0,Y 269.344,Z 496.288,A -85,B 0,C 180,E1 20124.873,E2 20124.873} C_VEL
LIN {X 0,Y 264.81,Z 485.212,A -85,B 0,C 180,E1 20128.597,E2 20128.597} C_VEL
LIN {X 0,Y 261.471,Z 477.64,A -85,B 0,C 180,E1 20131.446,E2 20131.446} C_VEL
LIN {X 0,Y 259.77,Z 473.857,A -85,B 0,C 180,E1 20132.988,E2 20132.988} C_VEL
LIN {X 0,Y 258.597,Z 470.647,A -85,B 0,C 180,E1 20134.459,E2 20134.459} C_VEL
LIN {X 0,Y 258.59,Z 470.554,A -85,B 0,C 180,E1 20139.399,E2 20139.399} C_VEL
LIN {X 0,Y 258.589,Z 470.544,A -85,B 0,C 180,E1 20144.321,E2 20144.321} C_VEL
LIN {X 0,Y 258.577,Z 470.574,A -85,B 0,C 180,E1 20149.304,E2 20149.304} C_VEL
LIN {X 0,Y 258.594,Z 470.558,A -85,B 0,C 180,E1 20154.231,E2 20154.231} C_VEL
LIN {X 0,Y 258.565,Z 470.536,A -85,B 0,C 180,E1 20159.114,E2 20159.114} C_VEL
LIN {X 0,Y 258.581,Z 470.584,A -85,B 0,C 180,E1 20163.992,E2 20163.992} C_VEL
LIN {X 0,Y 258.577,Z 470.525,A -85,B 0,C 180,E1 20168.674,E2 20168.674} C_VEL
LIN {X 0,Y 258.564,Z 470.588,A -85,B 0,C 180,E1 20173.644,E2 20173.644} C_VEL
LIN {X 0,Y 258.575,Z 470.53,A -85,B 0,C 180,E1 20178.487,E2 20178.487} C_VEL
LIN {X 0,Y 258.563,Z 470.574,A -85,B 0,C 180,E1 20183.231,E2 20183.231} C_VEL
LIN {X 0,Y 258.559,Z 470.551,A -85,B 0,C 180,E1 20188.153,E2 20188.153} C_VEL
LIN {X 0,Y 258.571,Z 470.546,A -85,B 0,C 180,E1 20192.953,E2 20192.953} C_VEL
LIN {X 0,Y 258.548,Z 470.593,A -85,B 0,C 180,E1 20197.944,E2 20197.944} C_VEL
LIN {X 0,Y 258.561,Z 470.558,A -85,B 0,C 180,E1 20202.891,E2 20202.891} C_VEL
LIN {X 0,Y 258.542,Z 470.557,A -85,B 0,C 180,E1 20207.707,E2 20207.707} C_VEL
LIN {X 0,Y 258.6,Z 470.888,A -85,B 0,C 180,E1 20211.472,E2 20211.472} C_VEL
LIN {X 0,Y 261.798,Z 478.919,A -85,B 0,C 180,E1 20215.048,E2 20215.048} C_VEL
LIN {X 0,Y 265.54,Z 488.701,A -85,B 0,C 180,E1 20218.945,E2 20218.945} C_VEL
LIN {X 0,Y 269.494,Z 500.362,A -85,B 0,C 180,E1 20223.087,E2 20223.087} C_VEL
LIN {X 0,Y 273.087,Z 512.468,A -85,B 0,C 180,E1 20226.935,E2 20226.935} C_VEL
LIN {X 0,Y 276.627,Z 526.581,A -85,B 0,C 180,E1 20231.016,E2 20231.016} C_VEL
LIN {X 0,Y 278.452,Z 535.123,A -85,B 0,C 180,E1 20233.305,E2 20233.305} C_VEL
LIN {X 0,Y 275.002,Z 552.129,A -85,B 0,C 180,E1 20236.658,E2 20236.658} C_VEL
LIN {X 0,Y 281.744,Z 600.317,A -85,B 0,C 180,E1 20238.999,E2 20238.999} C_VEL
LIN {X 0,Y 278.09,Z 688.832,A -85,B 0,C 180,E1 20241.347,E2 20241.347} C_VEL
LIN {X 0,Y 276.894,Z 706.223,A -85,B 0,C 180,E1 20242.217,E2 20242.217} C_VEL
LIN {X 0,Y 275.317,Z 721.11,A -85,B 0,C 180,E1 20243.326,E2 20243.326} C_VEL
LIN {X 0,Y 273.205,Z 736.232,A -85,B 0,C 180,E1 20244.855,E2 20244.855} C_VEL
LIN {X 0,Y 270.93,Z 749.549,A -85,B 0,C 180,E1 20246.614,E2 20246.614} C_VEL
LIN {X 0,Y 268.388,Z 762.62,A -85,B 0,C 180,E1 20248.827,E2 20248.827} C_VEL
LIN {X 0,Y 265.933,Z 774.042,A -85,B 0,C 180,E1 20251.292,E2 20251.292} C_VEL
LIN {X 0,Y 263.595,Z 784.372,A -85,B 0,C 180,E1 20254.133,E2 20254.133} C_VEL
LIN {X 0,Y 261.731,Z 792.526,A -85,B 0,C 180,E1 20257.021,E2 20257.021} C_VEL
LIN {X 0,Y 260.153,Z 799.765,A -85,B 0,C 180,E1 20260.406,E2 20260.406} C_VEL
LIN {X 0,Y 259.171,Z 804.977,A -85,B 0,C 180,E1 20263.838,E2 20263.838} C_VEL
LIN {X 0,Y 258.724,Z 808.59,A -85,B 0,C 180,E1 20267.544,E2 20267.544} C_VEL
LIN {X 0,Y 258.817,Z 810.185,A -85,B 0,C 180,E1 20271.055,E2 20271.055} C_VEL
LIN {X 0,Y 259.506,Z 810.09,A -85,B 0,C 180,E1 20274.832,E2 20274.832} C_VEL
LIN {X 0,Y 260.189,Z 809.145,A -85,B 0,C 180,E1 20276.958,E2 20276.958} C_VEL
LIN {X 0,Y 259.912,Z 808.151,A -85,B 0,C 180,E1 20278.656,E2 20278.656} C_VEL
LIN {X 0,Y 256.946,Z 805.476,A -85,B 0,C 180,E1 20282.272,E2 20282.272} C_VEL
LIN {X 0,Y 256.621,Z 803.146,A -85,B 0,C 180,E1 20284.184,E2 20284.184} C_VEL
LIN {X 0,Y 256.912,Z 802.391,A -85,B 0,C 180,E1 20284.646,E2 20284.646} C_VEL
LIN {X 0,Y 260.168,Z 795.7,A -85,B 0,C 180,E1 20288.015,E2 20288.015} C_VEL
LIN {X 0,Y 263.795,Z 787.486,A -85,B 0,C 180,E1 20291.038,E2 20291.038} C_VEL
LIN {X 0,Y 267.627,Z 777.99,A -85,B 0,C 180,E1 20293.722,E2 20293.722} C_VEL
LIN {X 0,Y 271.632,Z 766.812,A -85,B 0,C 180,E1 20296.175,E2 20296.175} C_VEL
LIN {X 0,Y 275.656,Z 754.013,A -85,B 0,C 180,E1 20298.348,E2 20298.348} C_VEL
LIN {X 0,Y 279.275,Z 740.327,A -85,B 0,C 180,E1 20300.144,E2 20300.144} C_VEL
LIN {X 0,Y 282.446,Z 725.394,A -85,B 0,C 180,E1 20301.638,E2 20301.638} C_VEL
LIN {X 0,Y 284.89,Z 710.022,A -85,B 0,C 180,E1 20302.773,E2 20302.773} C_VEL
LIN {X 0,Y 286.667,Z 692.948,A -85,B 0,C 180,E1 20303.629,E2 20303.629} C_VEL
LIN {X 0,Y 289.453,Z 646.661,A -85,B 0,C 180,E1 20304.919,E2 20304.919} C_VEL
LIN {X 0,Y 291.796,Z 605.43,A -85,B 0,C 180,E1 20305.986,E2 20305.986} C_VEL
LIN {X 0,Y 287.862,Z 578.321,A -85,B 0,C 180,E1 20307.897,E2 20307.897} C_VEL
